(* PLC project Adressering.ecp, WAGO e!COCKPIT e!COCKPIT *)
(* stored: creationDateTime 2021-01-18T14:20:23.2110188, modificationDateTime 2021-01-18T11:51:27.6823754 *)

TYPE dtRomtype_11111111 : STRUCT
  RB601_V : BOOL;  (* Bevegelse *)
  RB601_HVAC : BOOL;  (* HVAC signal *)
  RT601_CT : REAL;  (* Rom temperatur *)
  RT601_SP_D : REAL;  (* Temperatur SP *)
  RT601_SP_S : REAL;  (* Temperatur SP standby *)
  RT601_SP_N : REAL;  (* Temperatur SP nattsenk *)
  RT601_SP_F : REAL;  (* Temperatur SP frostsikring *)
  RT601_CS : REAL;  (* Aktivt temperatur SP *)
  OPM : INT;  (* Rom modus *)
  OPM_CV : INT;  (* Rom modus verdi *)
  RY601_CV : REAL;  (* Co2 Nivaa *)
  RY601_SP : REAL;  (* Co2 SP *)
  RY601_MAN : BOOL;  (* Co2 Man mode *)
  RY601_OP : REAL;  (* Co2 paadrag *)
  LH601_OP : REAL;  (* Varmepaadrag *)
  LH601_MAN : BOOL;  (* Force LH *)
  LH601_CMD : BOOL;  (* LH601_CMD *)
  LC601_OP : REAL;  (* LC601_OP *)
  LC601_SP : REAL;  (* LC SP *)
  LC601_MAN : BOOL;  (* Force LC *)
  LC601_CMD : BOOL;  (* LC601_CMD *)
END_STRUCT;
END_TYPE

TYPE dtRomtype_22111111 : STRUCT
  RB601_V : BOOL;  (* Bevegelse *)
  RB602_V : BOOL;  (* Bevegelse *)
  RB601_HVAC : BOOL;  (* HVAC signal *)
  RB602_HVAC : BOOL;  (* HVAC signal *)
  RB600_HVAC : BOOL;  (* HVAC signal samlet *)
  RT601_CT : REAL;  (* Rom temperatur *)
  RT601_SP_D : REAL;  (* Temperatur SP *)
  RT601_SP_S : REAL;  (* Temperatur SP standby *)
  RT601_SP_N : REAL;  (* Temperatur SP nattsenk *)
  RT601_SP_F : REAL;  (* Temperatur SP frostsikring *)
  RT601_CS : REAL;  (* Aktivt temperatur SP *)
  OPM : INT;  (* Rom modus *)
  OPM_CV : INT;  (* Rom modus verdi *)
  RY601_CV : REAL;  (* Co2 Nivaa *)
  RY601_SP : REAL;  (* Co2 SP *)
  RY601_MAN : BOOL;  (* Co2 Man mode *)
  RY601_OP : REAL;  (* Co2 paadrag *)
  LH601_OP : REAL;  (* Varmepaadrag *)
  LH601_MAN : BOOL;  (* Force LH *)
  LH601_CMD : BOOL;  (* LH601_CMD *)
  LC601_OP : REAL;  (* LC601_OP *)
  LC601_SP : REAL;  (* LC SP *)
  LC601_MAN : BOOL;  (* Force LC *)
  LC601_CMD : BOOL;  (* LC601_CMD *)
END_STRUCT;
END_TYPE

TYPE dtRomtype_11211111 : STRUCT
  RB601_V : BOOL;  (* Bevegelse *)
  RB601_HVAC : BOOL;  (* HVAC signal *)
  RT601_CT : REAL;  (* Rom temperatur *)
  RT602_CT : REAL;  (* Rom temperatur *)
  RT600_CT : REAL;  (* Temperatur SP *)
  RT600_SP_D : REAL;  (* Temperatur SP *)
  RT600_SP_S : REAL;  (* Temperatur SP standby *)
  RT600_SP_N : REAL;  (* Temperatur SP nattsenk *)
  RT600_SP_F : REAL;  (* Temperatur SP frostsikring *)
  RT600_CS : REAL;  (* Aktivt temperatur SP *)
  OPM : INT;  (* Rom modus *)
  OPM_CV : INT;  (* Rom modus verdi *)
  RY601_CV : REAL;  (* Co2 Nivaa *)
  RY601_SP : REAL;  (* Co2 SP *)
  RY601_MAN : BOOL;  (* Co2 Man mode *)
  RY601_OP : REAL;  (* Co2 paadrag *)
  LH601_OP : REAL;  (* Varmepaadrag *)
  LH601_MAN : BOOL;  (* Force LH *)
  LH601_CMD : BOOL;  (* LH601_CMD *)
  LC601_OP : REAL;  (* LC601_OP *)
  LC601_SP : REAL;  (* LC SP *)
  LC601_MAN : BOOL;  (* Force LC *)
  LC601_CMD : BOOL;  (* LC601_CMD *)
END_STRUCT;
END_TYPE

TYPE dtRomtype_11121111 : STRUCT
  RB601_V : BOOL;  (* Bevegelse *)
  RB601_HVAC : BOOL;  (* HVAC signal *)
  RT601_CT : REAL;  (* Rom temperatur *)
  RT601_SP_D : REAL;  (* Temperatur SP *)
  RT601_SP_S : REAL;  (* Temperatur SP standby *)
  RT601_SP_N : REAL;  (* Temperatur SP nattsenk *)
  RT601_SP_F : REAL;  (* Temperatur SP frostsikring *)
  RT601_CS : REAL;  (* Aktivt temperatur SP *)
  OPM : INT;  (* Rom modus *)
  OPM_CV : INT;  (* Rom modus verdi *)
  RY601_CV : REAL;  (* Co2 Nivaa *)
  RY602_CV : REAL;  (* Co2 Nivaa *)
  RY600_CV : REAL;  (* Co2 gjennomsnitt *)
  RY600_SP : REAL;  (* Co2 SP *)
  RY600_MAN : BOOL;  (* Co2 Man mode *)
  RY600_OP : REAL;  (* Co2 paadrag *)
  LH601_OP : REAL;  (* Varmepaadrag *)
  LH601_MAN : BOOL;  (* Force LH *)
  LH601_CMD : BOOL;  (* LH601_CMD *)
  LC601_OP : REAL;  (* LC601_OP *)
  LC601_SP : REAL;  (* LC SP *)
  LC601_MAN : BOOL;  (* Force LC *)
  LC601_CMD : BOOL;  (* LC601_CMD *)
END_STRUCT;
END_TYPE

TYPE dtRomtype_11112111 : STRUCT
  RB601_V : BOOL;  (* Bevegelse *)
  RB601_HVAC : BOOL;  (* HVAC signal *)
  RT601_CT : REAL;  (* Rom temperatur *)
  RT601_SP_D : REAL;  (* Temperatur SP *)
  RT601_SP_S : REAL;  (* Temperatur SP standby *)
  RT601_SP_N : REAL;  (* Temperatur SP nattsenk *)
  RT601_SP_F : REAL;  (* Temperatur SP frostsikring *)
  RT601_CS : REAL;  (* Aktivt temperatur SP *)
  OPM : INT;  (* Rom modus *)
  OPM_CV : INT;  (* Rom modus verdi *)
  RY601_CV : REAL;  (* Co2 Nivaa *)
  RY601_SP : REAL;  (* Co2 SP *)
  RY601_MAN : BOOL;  (* Co2 Man mode *)
  RY601_OP : REAL;  (* Co2 paadrag *)
  LH601_OP : REAL;  (* Varmepaadrag *)
  LH602_OP : REAL;  (* Varmepaadrag *)
  LH601_MAN : BOOL;  (* Force LH *)
  LH601_CMD : BOOL;  (* LH601_CMD *)
  LC601_OP : REAL;  (* LC601_OP *)
  LC601_SP : REAL;  (* LC SP *)
  LC601_MAN : BOOL;  (* Force LC *)
  LC601_CMD : BOOL;  (* LC601_CMD *)
END_STRUCT;
END_TYPE

TYPE dtRomtype_11111211 : STRUCT
  RB601_V : BOOL;  (* Bevegelse *)
  RB601_HVAC : BOOL;  (* HVAC signal *)
  RT601_CT : REAL;  (* Rom temperatur *)
  RT601_SP_D : REAL;  (* Temperatur SP *)
  RT601_SP_S : REAL;  (* Temperatur SP standby *)
  RT601_SP_N : REAL;  (* Temperatur SP nattsenk *)
  RT601_SP_F : REAL;  (* Temperatur SP frostsikring *)
  RT601_CS : REAL;  (* Aktivt temperatur SP *)
  OPM : INT;  (* Rom modus *)
  OPM_CV : INT;  (* Rom modus verdi *)
  RY601_CV : REAL;  (* Co2 Nivaa *)
  RY601_SP : REAL;  (* Co2 SP *)
  RY601_MAN : BOOL;  (* Co2 Man mode *)
  RY601_OP : REAL;  (* Co2 paadrag *)
  LH601_OP : REAL;  (* Varmepaadrag *)
  LH601_MAN : BOOL;  (* Force LH *)
  LH601_CMD : BOOL;  (* LH601_CMD *)
  LH602_CMD : BOOL;  (* LH602_CMD *)
  LC601_OP : REAL;  (* LC601_OP *)
  LC601_SP : REAL;  (* LC SP *)
  LC601_MAN : BOOL;  (* Force LC *)
  LC601_CMD : BOOL;  (* LC601_CMD *)
END_STRUCT;
END_TYPE

TYPE dtRomtype_11111121 : STRUCT
  RB601_V : BOOL;  (* Bevegelse *)
  RB601_HVAC : BOOL;  (* HVAC signal *)
  RT601_CT : REAL;  (* Rom temperatur *)
  RT601_SP_D : REAL;  (* Temperatur SP *)
  RT601_SP_S : REAL;  (* Temperatur SP standby *)
  RT601_SP_N : REAL;  (* Temperatur SP nattsenk *)
  RT601_SP_F : REAL;  (* Temperatur SP frostsikring *)
  RT601_CS : REAL;  (* Aktivt temperatur SP *)
  OPM : INT;  (* Rom modus *)
  OPM_CV : INT;  (* Rom modus verdi *)
  RY601_CV : REAL;  (* Co2 Nivaa *)
  RY601_SP : REAL;  (* Co2 SP *)
  RY601_MAN : BOOL;  (* Co2 Man mode *)
  RY601_OP : REAL;  (* Co2 paadrag *)
  LH601_OP : REAL;  (* Varmepaadrag *)
  LH601_MAN : BOOL;  (* Force LH *)
  LH601_CMD : BOOL;  (* LH601_CMD *)
  LC601_OP : REAL;  (* LC601_OP *)
  LC602_OP : REAL;  (* LC602_OP *)
  LC601_SP : REAL;  (* LC SP *)
  LC601_MAN : BOOL;  (* Force LC *)
  LC601_CMD : BOOL;  (* LC601_CMD *)
END_STRUCT;
END_TYPE

TYPE dtRomtype_11111112 : STRUCT
  RB601_V : BOOL;  (* Bevegelse *)
  RB601_HVAC : BOOL;  (* HVAC signal *)
  RT601_CT : REAL;  (* Rom temperatur *)
  RT601_SP_D : REAL;  (* Temperatur SP *)
  RT601_SP_S : REAL;  (* Temperatur SP standby *)
  RT601_SP_N : REAL;  (* Temperatur SP nattsenk *)
  RT601_SP_F : REAL;  (* Temperatur SP frostsikring *)
  RT601_CS : REAL;  (* Aktivt temperatur SP *)
  OPM : INT;  (* Rom modus *)
  OPM_CV : INT;  (* Rom modus verdi *)
  RY601_CV : REAL;  (* Co2 Nivaa *)
  RY601_SP : REAL;  (* Co2 SP *)
  RY601_MAN : BOOL;  (* Co2 Man mode *)
  RY601_OP : REAL;  (* Co2 paadrag *)
  LH601_OP : REAL;  (* Varmepaadrag *)
  LH601_MAN : BOOL;  (* Force LH *)
  LH601_CMD : BOOL;  (* LH601_CMD *)
  LC601_OP : REAL;  (* LC601_OP *)
  LC601_SP : REAL;  (* LC SP *)
  LC601_MAN : BOOL;  (* Force LC *)
  LC601_CMD : BOOL;  (* LC601_CMD *)
  LC602_CMD : BOOL;  (* LC602_CMD *)
END_STRUCT;
END_TYPE

TYPE dtRomtype_11212111 : STRUCT
  RB601_V : BOOL;  (* Bevegelse *)
  RB601_HVAC : BOOL;  (* HVAC signal *)
  RT601_CT : REAL;  (* Rom temperatur *)
  RT602_CT : REAL;  (* Rom temperatur *)
  RT600_CT : REAL;  (* Temperatur SP *)
  RT600_SP_D : REAL;  (* Temperatur SP *)
  RT600_SP_S : REAL;  (* Temperatur SP standby *)
  RT600_SP_N : REAL;  (* Temperatur SP nattsenk *)
  RT600_SP_F : REAL;  (* Temperatur SP frostsikring *)
  RT600_CS : REAL;  (* Aktivt temperatur SP *)
  OPM : INT;  (* Rom modus *)
  OPM_CV : INT;  (* Rom modus verdi *)
  RY601_CV : REAL;  (* Co2 Nivaa *)
  RY601_SP : REAL;  (* Co2 SP *)
  RY601_MAN : BOOL;  (* Co2 Man mode *)
  RY601_OP : REAL;  (* Co2 paadrag *)
  LH601_OP : REAL;  (* Varmepaadrag *)
  LH602_OP : REAL;  (* Varmepaadrag *)
  LH601_MAN : BOOL;  (* Force LH *)
  LH601_CMD : BOOL;  (* LH601_CMD *)
  LC601_OP : REAL;  (* LC601_OP *)
  LC601_SP : REAL;  (* LC SP *)
  LC601_MAN : BOOL;  (* Force LC *)
  LC601_CMD : BOOL;  (* LC601_CMD *)
END_STRUCT;
END_TYPE

TYPE dtRomtype_11211211 : STRUCT
  RB601_V : BOOL;  (* Bevegelse *)
  RB601_HVAC : BOOL;  (* HVAC signal *)
  RT601_CT : REAL;  (* Rom temperatur *)
  RT602_CT : REAL;  (* Rom temperatur *)
  RT600_CT : REAL;  (* Temperatur SP *)
  RT600_SP_D : REAL;  (* Temperatur SP *)
  RT600_SP_S : REAL;  (* Temperatur SP standby *)
  RT600_SP_N : REAL;  (* Temperatur SP nattsenk *)
  RT600_SP_F : REAL;  (* Temperatur SP frostsikring *)
  RT600_CS : REAL;  (* Aktivt temperatur SP *)
  OPM : INT;  (* Rom modus *)
  OPM_CV : INT;  (* Rom modus verdi *)
  RY601_CV : REAL;  (* Co2 Nivaa *)
  RY601_SP : REAL;  (* Co2 SP *)
  RY601_MAN : BOOL;  (* Co2 Man mode *)
  RY601_OP : REAL;  (* Co2 paadrag *)
  LH601_OP : REAL;  (* Varmepaadrag *)
  LH601_MAN : BOOL;  (* Force LH *)
  LH601_CMD : BOOL;  (* LH601_CMD *)
  LH602_CMD : BOOL;  (* LH602_CMD *)
  LC601_OP : REAL;  (* LC601_OP *)
  LC601_SP : REAL;  (* LC SP *)
  LC601_MAN : BOOL;  (* Force LC *)
  LC601_CMD : BOOL;  (* LC601_CMD *)
END_STRUCT;
END_TYPE

TYPE dtRomtype_11211121 : STRUCT
  RB601_V : BOOL;  (* Bevegelse *)
  RB601_HVAC : BOOL;  (* HVAC signal *)
  RT601_CT : REAL;  (* Rom temperatur *)
  RT602_CT : REAL;  (* Rom temperatur *)
  RT600_CT : REAL;  (* Temperatur SP *)
  RT600_SP_D : REAL;  (* Temperatur SP *)
  RT600_SP_S : REAL;  (* Temperatur SP standby *)
  RT600_SP_N : REAL;  (* Temperatur SP nattsenk *)
  RT600_SP_F : REAL;  (* Temperatur SP frostsikring *)
  RT600_CS : REAL;  (* Aktivt temperatur SP *)
  OPM : INT;  (* Rom modus *)
  OPM_CV : INT;  (* Rom modus verdi *)
  RY601_CV : REAL;  (* Co2 Nivaa *)
  RY601_SP : REAL;  (* Co2 SP *)
  RY601_MAN : BOOL;  (* Co2 Man mode *)
  RY601_OP : REAL;  (* Co2 paadrag *)
  LH601_OP : REAL;  (* Varmepaadrag *)
  LH601_MAN : BOOL;  (* Force LH *)
  LH601_CMD : BOOL;  (* LH601_CMD *)
  LC601_OP : REAL;  (* LC601_OP *)
  LC602_OP : REAL;  (* LC602_OP *)
  LC601_SP : REAL;  (* LC SP *)
  LC601_MAN : BOOL;  (* Force LC *)
  LC601_CMD : BOOL;  (* LC601_CMD *)
END_STRUCT;
END_TYPE

TYPE dtRomtype_11211112 : STRUCT
  RB601_V : BOOL;  (* Bevegelse *)
  RB601_HVAC : BOOL;  (* HVAC signal *)
  RT601_CT : REAL;  (* Rom temperatur *)
  RT602_CT : REAL;  (* Rom temperatur *)
  RT600_CT : REAL;  (* Temperatur SP *)
  RT600_SP_D : REAL;  (* Temperatur SP *)
  RT600_SP_S : REAL;  (* Temperatur SP standby *)
  RT600_SP_N : REAL;  (* Temperatur SP nattsenk *)
  RT600_SP_F : REAL;  (* Temperatur SP frostsikring *)
  RT600_CS : REAL;  (* Aktivt temperatur SP *)
  OPM : INT;  (* Rom modus *)
  OPM_CV : INT;  (* Rom modus verdi *)
  RY601_CV : REAL;  (* Co2 Nivaa *)
  RY601_SP : REAL;  (* Co2 SP *)
  RY601_MAN : BOOL;  (* Co2 Man mode *)
  RY601_OP : REAL;  (* Co2 paadrag *)
  LH601_OP : REAL;  (* Varmepaadrag *)
  LH601_MAN : BOOL;  (* Force LH *)
  LH601_CMD : BOOL;  (* LH601_CMD *)
  LC601_OP : REAL;  (* LC601_OP *)
  LC601_SP : REAL;  (* LC SP *)
  LC601_MAN : BOOL;  (* Force LC *)
  LC601_CMD : BOOL;  (* LC601_CMD *)
  LC602_CMD : BOOL;  (* LC602_CMD *)
END_STRUCT;
END_TYPE

TYPE dtRomtype_11221111 : STRUCT
  RB601_V : BOOL;  (* Bevegelse *)
  RB601_HVAC : BOOL;  (* HVAC signal *)
  RT601_CT : REAL;  (* Rom temperatur *)
  RT602_CT : REAL;  (* Rom temperatur *)
  RT600_CT : REAL;  (* Temperatur SP *)
  RT600_SP_D : REAL;  (* Temperatur SP *)
  RT600_SP_S : REAL;  (* Temperatur SP standby *)
  RT600_SP_N : REAL;  (* Temperatur SP nattsenk *)
  RT600_SP_F : REAL;  (* Temperatur SP frostsikring *)
  RT600_CS : REAL;  (* Aktivt temperatur SP *)
  OPM : INT;  (* Rom modus *)
  OPM_CV : INT;  (* Rom modus verdi *)
  RY601_CV : REAL;  (* Co2 Nivaa *)
  RY602_CV : REAL;  (* Co2 Nivaa *)
  RY600_CV : REAL;  (* Co2 gjennomsnitt *)
  RY600_SP : REAL;  (* Co2 SP *)
  RY600_MAN : BOOL;  (* Co2 Man mode *)
  RY600_OP : REAL;  (* Co2 paadrag *)
  LH601_OP : REAL;  (* Varmepaadrag *)
  LH601_MAN : BOOL;  (* Force LH *)
  LH601_CMD : BOOL;  (* LH601_CMD *)
  LC601_OP : REAL;  (* LC601_OP *)
  LC601_SP : REAL;  (* LC SP *)
  LC601_MAN : BOOL;  (* Force LC *)
  LC601_CMD : BOOL;  (* LC601_CMD *)
END_STRUCT;
END_TYPE

TYPE dtRomtype_11222222 : STRUCT
  RB601_V : BOOL;  (* Bevegelse *)
  RB601_HVAC : BOOL;  (* HVAC signal *)
  RT601_CT : REAL;  (* Rom temperatur *)
  RT602_CT : REAL;  (* Rom temperatur *)
  RT600_CT : REAL;  (* Temperatur SP *)
  RT600_SP_D : REAL;  (* Temperatur SP *)
  RT600_SP_S : REAL;  (* Temperatur SP standby *)
  RT600_SP_N : REAL;  (* Temperatur SP nattsenk *)
  RT600_SP_F : REAL;  (* Temperatur SP frostsikring *)
  RT600_CS : REAL;  (* Aktivt temperatur SP *)
  OPM : INT;  (* Rom modus *)
  OPM_CV : INT;  (* Rom modus verdi *)
  RY601_CV : REAL;  (* Co2 Nivaa *)
  RY602_CV : REAL;  (* Co2 Nivaa *)
  RY600_CV : REAL;  (* Co2 gjennomsnitt *)
  RY600_SP : REAL;  (* Co2 SP *)
  RY600_MAN : BOOL;  (* Co2 Man mode *)
  RY600_OP : REAL;  (* Co2 paadrag *)
  LH601_OP : REAL;  (* Varmepaadrag *)
  LH602_OP : REAL;  (* Varmepaadrag *)
  LH601_MAN : BOOL;  (* Force LH *)
  LH601_CMD : BOOL;  (* LH601_CMD *)
  LH602_CMD : BOOL;  (* LH602_CMD *)
  LC601_OP : REAL;  (* LC601_OP *)
  LC602_OP : REAL;  (* LC602_OP *)
  LC601_SP : REAL;  (* LC SP *)
  LC601_MAN : BOOL;  (* Force LC *)
  LC601_CMD : BOOL;  (* LC601_CMD *)
  LC602_CMD : BOOL;  (* LC602_CMD *)
END_STRUCT;
END_TYPE

TYPE dtRomtype_22222222 : STRUCT
  RB601_V : BOOL;  (* Bevegelse *)
  RB602_V : BOOL;  (* Bevegelse *)
  RB601_HVAC : BOOL;  (* HVAC signal *)
  RB602_HVAC : BOOL;  (* HVAC signal *)
  RB600_HVAC : BOOL;  (* HVAC signal samlet *)
  RT601_CT : REAL;  (* Rom temperatur *)
  RT602_CT : REAL;  (* Rom temperatur *)
  RT600_CT : REAL;  (* Temperatur SP *)
  RT600_SP_D : REAL;  (* Temperatur SP *)
  RT600_SP_S : REAL;  (* Temperatur SP standby *)
  RT600_SP_N : REAL;  (* Temperatur SP nattsenk *)
  RT600_SP_F : REAL;  (* Temperatur SP frostsikring *)
  RT600_CS : REAL;  (* Aktivt temperatur SP *)
  OPM : INT;  (* Rom modus *)
  OPM_CV : INT;  (* Rom modus verdi *)
  RY601_CV : REAL;  (* Co2 Nivaa *)
  RY602_CV : REAL;  (* Co2 Nivaa *)
  RY600_CV : REAL;  (* Co2 gjennomsnitt *)
  RY600_SP : REAL;  (* Co2 SP *)
  RY600_MAN : BOOL;  (* Co2 Man mode *)
  RY600_OP : REAL;  (* Co2 paadrag *)
  LH601_OP : REAL;  (* Varmepaadrag *)
  LH602_OP : REAL;  (* Varmepaadrag *)
  LH601_MAN : BOOL;  (* Force LH *)
  LH601_CMD : BOOL;  (* LH601_CMD *)
  LH602_CMD : BOOL;  (* LH602_CMD *)
  LC601_OP : REAL;  (* LC601_OP *)
  LC602_OP : REAL;  (* LC602_OP *)
  LC601_SP : REAL;  (* LC SP *)
  LC601_MAN : BOOL;  (* Force LC *)
  LC601_CMD : BOOL;  (* LC601_CMD *)
  LC602_CMD : BOOL;  (* LC602_CMD *)
END_STRUCT;
END_TYPE

TYPE dtRomtype_22022222 : STRUCT
  RB601_V : BOOL;  (* Bevegelse *)
  RB602_V : BOOL;  (* Bevegelse *)
  RB601_HVAC : BOOL;  (* HVAC signal *)
  RB602_HVAC : BOOL;  (* HVAC signal *)
  RB600_HVAC : BOOL;  (* HVAC signal samlet *)
  RY601_CV : REAL;  (* Co2 Nivaa *)
  RY602_CV : REAL;  (* Co2 Nivaa *)
  RY600_CV : REAL;  (* Co2 gjennomsnitt *)
  RY600_SP : REAL;  (* Co2 SP *)
  RY600_MAN : BOOL;  (* Co2 Man mode *)
  RY600_OP : REAL;  (* Co2 paadrag *)
  LH601_OP : REAL;  (* Varmepaadrag *)
  LH602_OP : REAL;  (* Varmepaadrag *)
  LH601_MAN : BOOL;  (* Force LH *)
  LH601_CMD : BOOL;  (* LH601_CMD *)
  LH602_CMD : BOOL;  (* LH602_CMD *)
  LC601_OP : REAL;  (* LC601_OP *)
  LC602_OP : REAL;  (* LC602_OP *)
  LC601_SP : REAL;  (* LC SP *)
  LC601_MAN : BOOL;  (* Force LC *)
  LC601_CMD : BOOL;  (* LC601_CMD *)
  LC602_CMD : BOOL;  (* LC602_CMD *)
END_STRUCT;
END_TYPE

{attribute 'qualified_only'}
VAR_GLOBAL  (* STLV59_563 *)
  STLV59_A_563_RB001_HVAC : BOOL;  (* HVAC signal for PLS *)
  STLV59_A_563_KNX_Card_1_Status : BOOL;  (* KNX kort 1 status *)
  STLV59_A_563_001 : dtRomtype_11111111;  (* Test 1 *)
  STLV59_A_563_002 : dtRomtype_22111111;  (* Test 2 *)
  STLV59_A_563_003 : dtRomtype_11211111;  (* Test 3 *)
  STLV59_A_563_004 : dtRomtype_11121111;  (* Test 4 *)
  STLV59_A_563_005 : dtRomtype_11112111;  (* Test 5 *)
  STLV59_A_563_006 : dtRomtype_11111211;  (* Test 6 *)
  STLV59_A_563_007 : dtRomtype_11111121;  (* Test 7 *)
  STLV59_A_563_008 : dtRomtype_11111112;  (* Test 8 *)
  STLV59_A_563_009 : dtRomtype_11212111;  (* Test 9 *)
  STLV59_A_563_010 : dtRomtype_11211211;  (* Test 10 *)
  STLV59_A_563_011 : dtRomtype_11211121;  (* Test 11 *)
  STLV59_A_563_012 : dtRomtype_11211112;  (* Test 12 *)
  STLV59_A_563_013 : dtRomtype_11221111;  (* Test 13 *)
  STLV59_A_563_014 : dtRomtype_11222222;  (* Test 14 *)
  STLV59_A_563_015 : dtRomtype_22222222;  (* Test 15 *)
  STLV59_A_563_016 : dtRomtype_22022222;  (* Test 16 *)
END_VAR

FUNCTION_BLOCK fbRomtype_11111111
  VAR_INPUT
    RB601_HVAC : BOOL;
    RT601_CT : REAL;
    RT601_SP_D : REAL;
    RT601_SP_S : REAL;
    RT601_SP_N : REAL;
    RT601_SP_F : REAL;
    OPM : INT;
    RY601_CV : REAL;
    RY601_SP : REAL;
    RY601_MAN : BOOL;
    LH601_MAN : BOOL;
    LC601_SP : REAL;
    LC601_MAN : BOOL;
  END_VAR
  VAR
    RY601_PID_Man : BOOL;  (* Co2 regulering *)
    RY601_PID_ManVal : REAL;
    RY601_PID : fbSE_PID;
    RY601_PID_Kp : REAL := 1;  (* PID Luft rom. Forsterkning *)
    RY601_PID_Ti : REAL := 10;  (* PID luft rom. I-tid *)
    RY601_PID_Td : REAL;  (* PID luft rom. D-tid *)
    RY601_PID_Zero : REAL;  (* PID luft rom. 0-punkt *)
    RY601_PID_Max : REAL := 2000;  (* PID luft rom. Max verdi ppm *)
    RY601_PID_fMan : REAL := 100;  (* PID varme rom. Manuelt kjoeling *)
    LH601_PID : fbSE_PID;  (* PID varme rom *)
    LH601_PID_Kp : REAL := 1;  (* PID varme rom. Forsterkning *)
    LH601_PID_Ti : REAL := 10;  (* PID varme rom. I-tid *)
    LH601_PID_Td : REAL;  (* PID varme rom. D-tid *)
    LH601_PID_fMan : REAL := 100;  (* PID varme rom. Manuelt paadrag *)
    LH601_T : fbSE_Hyst;  (* Termostat varme rom *)
    LH601_T_On : REAL := 0.5;
    LH601_T_Off : REAL := 0.1;
    LC601_PID : fbSE_PID;  (* PID kjoeling rom *)
    LC601_PID_Kp : REAL := 1;  (* PID kjoeling rom. Forsterkning *)
    LC601_PID_Ti : REAL := 10;  (* PID kjoeling rom. I-tid *)
    LC601_PID_Td : REAL;  (* PID kjoeling rom. D-tid *)
    LC601_PID_fMan : REAL := 100;  (* PID varme rom. Manuelt kjoeling *)
    LC601_T : fbSE_Hyst;  (* Termostat kjoeling rom *)
    LC601_T_On : REAL := 0.5;
    LC601_T_Off : REAL := 0.1;
  END_VAR
  VAR_OUTPUT
    OPM_CV : INT;
    RT601_CS : REAL;
    RY601_OP : REAL;
    LH601_OP : REAL;
    LH601_CMD : BOOL;
    LC601_OP : REAL;
    LC601_CMD : BOOL;
  END_VAR

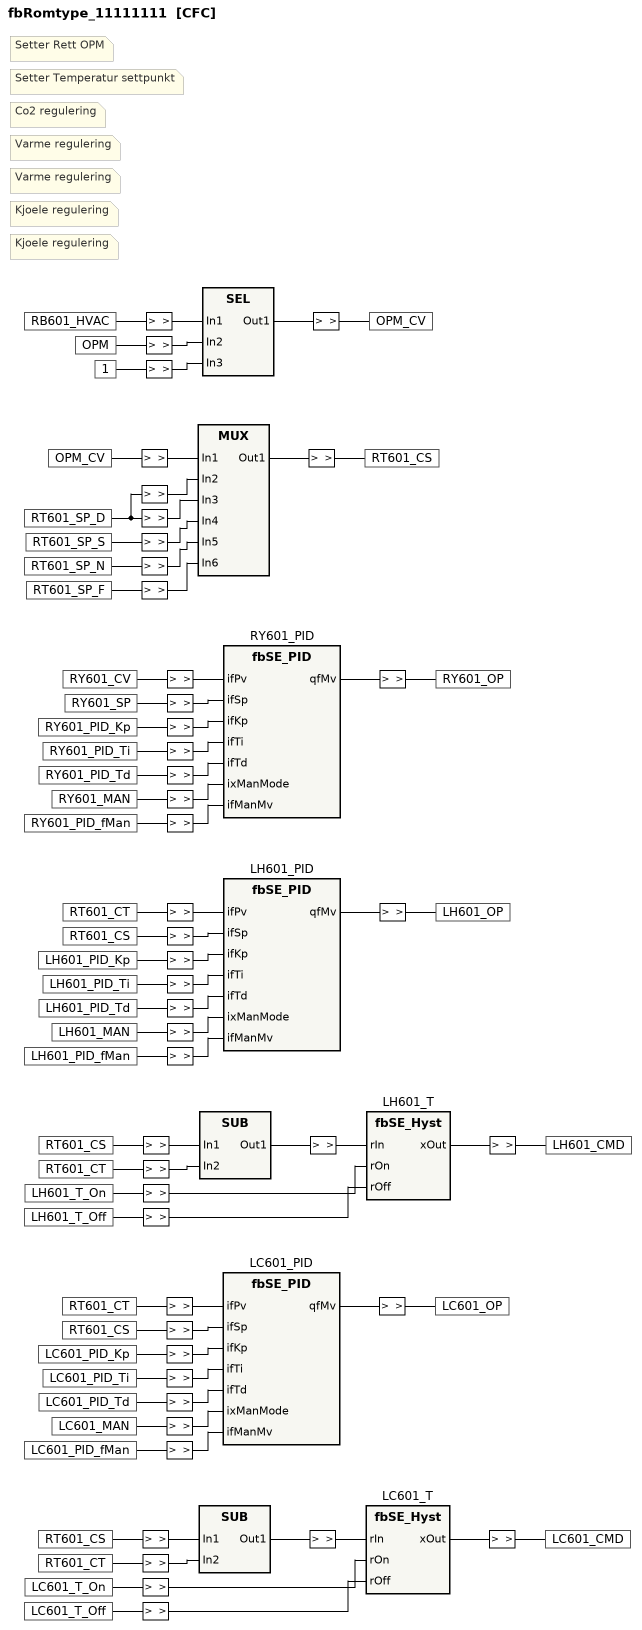
(* CFC diagram, written out as Structured Text *)
(* Setter Rett OPM *)
OPM_CV := SEL(RB601_HVAC, OPM, 1);
(* Setter Temperatur settpunkt *)
RT601_CS := MUX(OPM_CV, RT601_SP_D, RT601_SP_D, RT601_SP_S, RT601_SP_N, RT601_SP_F);
(* Co2 regulering *)
RY601_PID(ifPv := RY601_CV, ifSp := RY601_SP, ifKp := RY601_PID_Kp, ifTi := RY601_PID_Ti, ifTd := RY601_PID_Td, ixManMode := RY601_MAN, ifManMv := RY601_PID_fMan);
RY601_OP := RY601_PID.qfMv;
(* Varme regulering *)
LH601_PID(ifPv := RT601_CT, ifSp := RT601_CS, ifKp := LH601_PID_Kp, ifTi := LH601_PID_Ti, ifTd := LH601_PID_Td, ixManMode := LH601_MAN, ifManMv := LH601_PID_fMan);
LH601_OP := LH601_PID.qfMv;
(* Varme regulering *)
LH601_T(rIn := RT601_CS - RT601_CT, rOn := LH601_T_On, rOff := LH601_T_Off);
LH601_CMD := LH601_T.xOut;
(* Kjoele regulering *)
LC601_PID(ifPv := RT601_CT, ifSp := RT601_CS, ifKp := LC601_PID_Kp, ifTi := LC601_PID_Ti, ifTd := LC601_PID_Td, ixManMode := LC601_MAN, ifManMv := LC601_PID_fMan);
LC601_OP := LC601_PID.qfMv;
(* Kjoele regulering *)
LC601_T(rIn := RT601_CS - RT601_CT, rOn := LC601_T_On, rOff := LC601_T_Off);
LC601_CMD := LC601_T.xOut;
END_FUNCTION_BLOCK

FUNCTION_BLOCK fbRomtype_22111111
  VAR_INPUT
    RB601_HVAC : BOOL;
    RB602_HVAC : BOOL;
    RT601_CT : REAL;
    RT601_SP_D : REAL;
    RT601_SP_S : REAL;
    RT601_SP_N : REAL;
    RT601_SP_F : REAL;
    OPM : INT;
    RY601_CV : REAL;
    RY601_SP : REAL;
    RY601_MAN : BOOL;
    LH601_MAN : BOOL;
    LC601_SP : REAL;
    LC601_MAN : BOOL;
  END_VAR
  VAR
    RY601_PID_Man : BOOL;  (* Co2 regulering *)
    RY601_PID_ManVal : REAL;
    RY601_PID : fbSE_PID;
    RY601_PID_Kp : REAL := 1;  (* PID Luft rom. Forsterkning *)
    RY601_PID_Ti : REAL := 10;  (* PID luft rom. I-tid *)
    RY601_PID_Td : REAL;  (* PID luft rom. D-tid *)
    RY601_PID_Zero : REAL;  (* PID luft rom. 0-punkt *)
    RY601_PID_Max : REAL := 2000;  (* PID luft rom. Max verdi ppm *)
    RY601_PID_fMan : REAL := 100;  (* PID varme rom. Manuelt kjoeling *)
    LH601_PID : fbSE_PID;  (* PID varme rom *)
    LH601_PID_Kp : REAL := 1;  (* PID varme rom. Forsterkning *)
    LH601_PID_Ti : REAL := 10;  (* PID varme rom. I-tid *)
    LH601_PID_Td : REAL;  (* PID varme rom. D-tid *)
    LH601_PID_fMan : REAL := 100;  (* PID varme rom. Manuelt paadrag *)
    LH601_T : fbSE_Hyst;  (* Termostat varme rom *)
    LH601_T_On : REAL := 0.5;
    LH601_T_Off : REAL := 0.1;
    LC601_PID : fbSE_PID;  (* PID kjoeling rom *)
    LC601_PID_Kp : REAL := 1;  (* PID kjoeling rom. Forsterkning *)
    LC601_PID_Ti : REAL := 10;  (* PID kjoeling rom. I-tid *)
    LC601_PID_Td : REAL;  (* PID kjoeling rom. D-tid *)
    LC601_PID_fMan : REAL := 100;  (* PID varme rom. Manuelt kjoeling *)
    LC601_T : fbSE_Hyst;  (* Termostat kjoeling rom *)
    LC601_T_On : REAL := 0.5;
    LC601_T_Off : REAL := 0.1;
  END_VAR
  VAR_OUTPUT
    RB600_HVAC : BOOL;
    OPM_CV : INT;
    RT601_CS : REAL;
    RY601_OP : REAL;
    LH601_OP : REAL;
    LH601_CMD : BOOL;
    LC601_OP : REAL;
    LC601_CMD : BOOL;
  END_VAR
  VAR  (* added by the conversion: wires and edge detectors of the diagram *)
    _OR5_OUT : BOOL;
  END_VAR

(* CFC diagram, written out as Structured Text *)
(* Setter Rett OPM *)
_OR5_OUT := RB601_HVAC OR RB602_HVAC;
OPM_CV := SEL(_OR5_OUT, OPM, 1);
RB600_HVAC := _OR5_OUT;
(* Setter Temperatur settpunkt *)
RT601_CS := MUX(OPM_CV, RT601_SP_D, RT601_SP_D, RT601_SP_S, RT601_SP_N, RT601_SP_F);
(* Co2 regulering *)
RY601_PID(ifPv := RY601_CV, ifSp := RY601_SP, ifKp := RY601_PID_Kp, ifTi := RY601_PID_Ti, ifTd := RY601_PID_Td, ixManMode := RY601_MAN, ifManMv := RY601_PID_fMan);
RY601_OP := RY601_PID.qfMv;
(* Varme regulering *)
LH601_PID(ifPv := RT601_CT, ifSp := RT601_CS, ifKp := LH601_PID_Kp, ifTi := LH601_PID_Ti, ifTd := LH601_PID_Td, ixManMode := LH601_MAN, ifManMv := LH601_PID_fMan);
LH601_OP := LH601_PID.qfMv;
(* Varme regulering *)
LH601_T(rIn := RT601_CS - RT601_CT, rOn := LH601_T_On, rOff := LH601_T_Off);
LH601_CMD := LH601_T.xOut;
(* Kjoele regulering *)
LC601_PID(ifPv := RT601_CT, ifSp := RT601_CS, ifKp := LC601_PID_Kp, ifTi := LC601_PID_Ti, ifTd := LC601_PID_Td, ixManMode := LC601_MAN, ifManMv := LC601_PID_fMan);
LC601_OP := LC601_PID.qfMv;
(* Kjoele regulering *)
LC601_T(rIn := RT601_CS - RT601_CT, rOn := LC601_T_On, rOff := LC601_T_Off);
LC601_CMD := LC601_T.xOut;
END_FUNCTION_BLOCK

FUNCTION_BLOCK fbRomtype_11211111
  VAR_INPUT
    RB601_HVAC : BOOL;
    RT601_CT : REAL;
    RT602_CT : REAL;
    RT600_SP_D : REAL;
    RT600_SP_S : REAL;
    RT600_SP_N : REAL;
    RT600_SP_F : REAL;
    OPM : INT;
    RY601_CV : REAL;
    RY601_SP : REAL;
    RY601_MAN : BOOL;
    LH600_MAN : BOOL;
    LC600_SP : REAL;
    LC600_MAN : BOOL;
  END_VAR
  VAR
    RY601_PID_Man : BOOL;  (* Co2 regulering *)
    RY601_PID_ManVal : REAL;
    RY601_PID : fbSE_PID;
    RY601_PID_Kp : REAL := 1;  (* PID Luft rom. Forsterkning *)
    RY601_PID_Ti : REAL := 10;  (* PID luft rom. I-tid *)
    RY601_PID_Td : REAL;  (* PID luft rom. D-tid *)
    RY601_PID_Zero : REAL;  (* PID luft rom. 0-punkt *)
    RY601_PID_Max : REAL := 2000;  (* PID luft rom. Max verdi ppm *)
    RY601_PID_fMan : REAL := 100;  (* PID varme rom. Manuelt kjoeling *)
    LH600_PID : fbSE_PID;  (* PID varme rom *)
    LH600_PID_Kp : REAL := 1;  (* PID varme rom. Forsterkning *)
    LH600_PID_Ti : REAL := 10;  (* PID varme rom. I-tid *)
    LH600_PID_Td : REAL;  (* PID varme rom. D-tid *)
    LH600_PID_fMan : REAL := 100;  (* PID varme rom. Manuelt paadrag *)
    LH600_T : fbSE_Hyst;  (* Termostat varme rom *)
    LH600_T_On : REAL := 0.5;
    LH600_T_Off : REAL := 0.1;
    LC600_PID : fbSE_PID;  (* PID kjoeling rom *)
    LC600_PID_Kp : REAL := 1;  (* PID kjoeling rom. Forsterkning *)
    LC600_PID_Ti : REAL := 10;  (* PID kjoeling rom. I-tid *)
    LC600_PID_Td : REAL;  (* PID kjoeling rom. D-tid *)
    LC600_PID_fMan : REAL := 100;  (* PID varme rom. Manuelt kjoeling *)
    LC600_T : fbSE_Hyst;  (* Termostat kjoeling rom *)
    LC600_T_On : REAL := 0.5;
    LC600_T_Off : REAL := 0.1;
  END_VAR
  VAR_OUTPUT
    OPM_CV : INT;
    RT600_CT : REAL;
    RT600_CS : REAL;
    RY601_OP : REAL;
    LH601_OP : REAL;
    LH601_CMD : BOOL;
    LC601_OP : REAL;
    LC601_CMD : BOOL;
  END_VAR
  VAR  (* added by the conversion: wires and edge detectors of the diagram *)
    _ADD30_OUT : REAL;
    _DIV39_ENO : BOOL;
    _DIV39_OUT : REAL;
  END_VAR

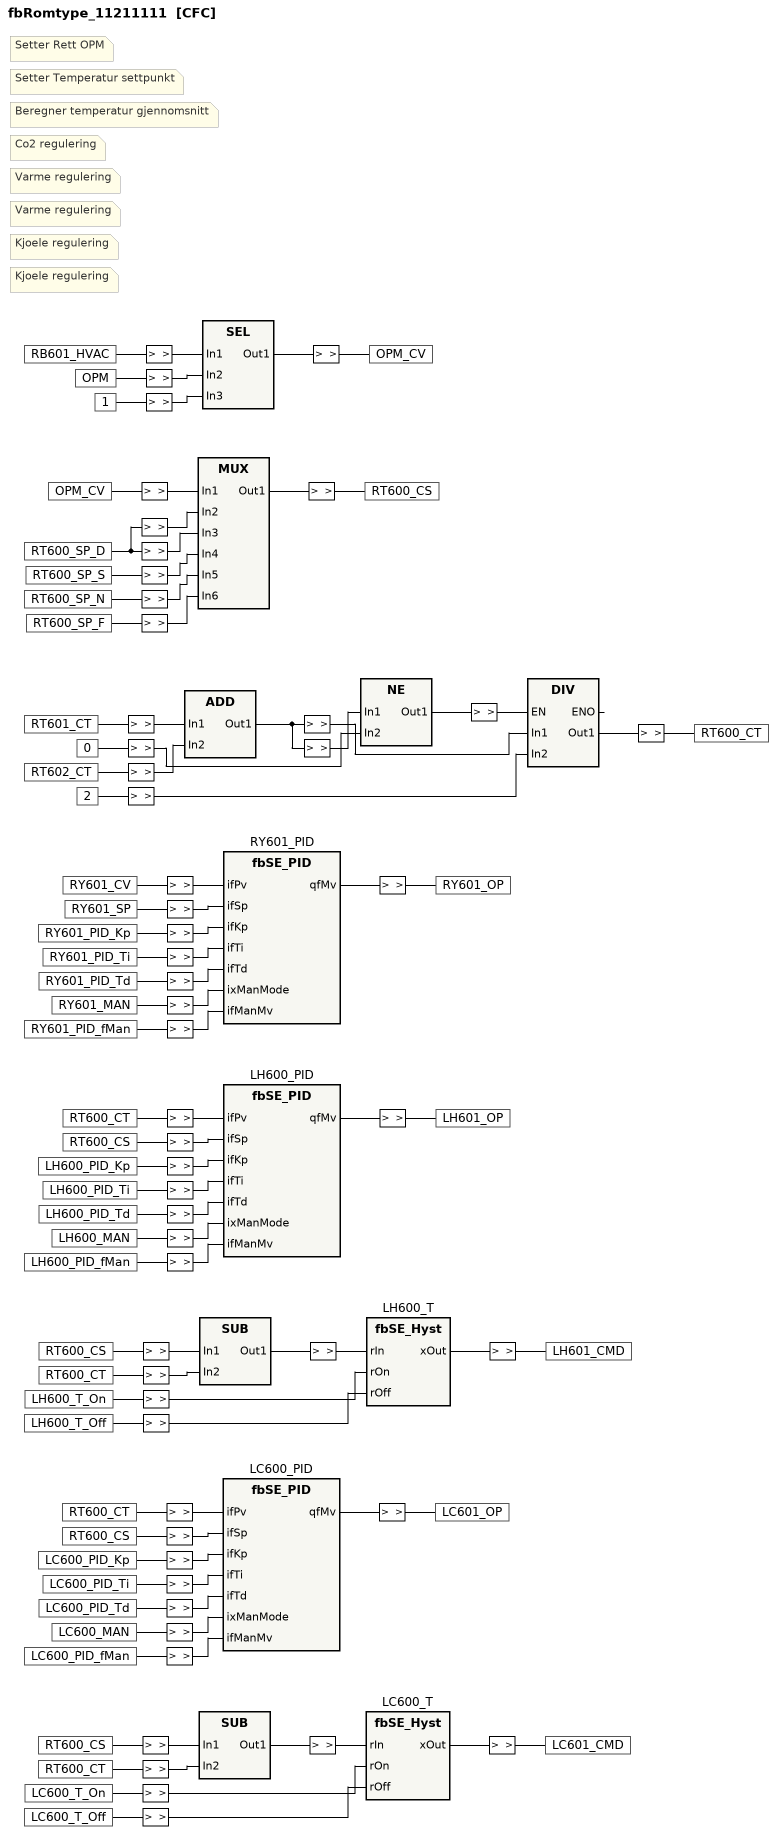
(* CFC diagram, written out as Structured Text *)
(* Setter Rett OPM *)
OPM_CV := SEL(RB601_HVAC, OPM, 1);
(* Setter Temperatur settpunkt *)
RT600_CS := MUX(OPM_CV, RT600_SP_D, RT600_SP_D, RT600_SP_S, RT600_SP_N, RT600_SP_F);
(* Beregner temperatur gjennomsnitt *)
_ADD30_OUT := RT601_CT + RT602_CT;
_DIV39_OUT := DIV(EN := _ADD30_OUT <> 0, IN1 := _ADD30_OUT, IN2 := 2, ENO => _DIV39_ENO);
IF _DIV39_ENO THEN RT600_CT := _DIV39_OUT; END_IF;
(* Co2 regulering *)
RY601_PID(ifPv := RY601_CV, ifSp := RY601_SP, ifKp := RY601_PID_Kp, ifTi := RY601_PID_Ti, ifTd := RY601_PID_Td, ixManMode := RY601_MAN, ifManMv := RY601_PID_fMan);
RY601_OP := RY601_PID.qfMv;
(* Varme regulering *)
LH600_PID(ifPv := RT600_CT, ifSp := RT600_CS, ifKp := LH600_PID_Kp, ifTi := LH600_PID_Ti, ifTd := LH600_PID_Td, ixManMode := LH600_MAN, ifManMv := LH600_PID_fMan);
LH601_OP := LH600_PID.qfMv;
(* Varme regulering *)
LH600_T(rIn := RT600_CS - RT600_CT, rOn := LH600_T_On, rOff := LH600_T_Off);
LH601_CMD := LH600_T.xOut;
(* Kjoele regulering *)
LC600_PID(ifPv := RT600_CT, ifSp := RT600_CS, ifKp := LC600_PID_Kp, ifTi := LC600_PID_Ti, ifTd := LC600_PID_Td, ixManMode := LC600_MAN, ifManMv := LC600_PID_fMan);
LC601_OP := LC600_PID.qfMv;
(* Kjoele regulering *)
LC600_T(rIn := RT600_CS - RT600_CT, rOn := LC600_T_On, rOff := LC600_T_Off);
LC601_CMD := LC600_T.xOut;
END_FUNCTION_BLOCK

FUNCTION_BLOCK fbRomtype_11121111
  VAR_INPUT
    RB601_HVAC : BOOL;
    RT601_CT : REAL;
    RT601_SP_D : REAL;
    RT601_SP_S : REAL;
    RT601_SP_N : REAL;
    RT601_SP_F : REAL;
    OPM : INT;
    RY601_CV : REAL;
    RY602_CV : REAL;
    RY600_SP : REAL;
    RY600_MAN : BOOL;
    LH601_MAN : BOOL;
    LC601_SP : REAL;
    LC601_MAN : BOOL;
  END_VAR
  VAR
    RY600_PID_Man : BOOL;  (* Co2 regulering *)
    RY600_PID_ManVal : REAL;
    RY600_PID : fbSE_PID;
    RY600_PID_Kp : REAL := 1;  (* PID Luft rom. Forsterkning *)
    RY600_PID_Ti : REAL := 10;  (* PID luft rom. I-tid *)
    RY600_PID_Td : REAL;  (* PID luft rom. D-tid *)
    RY600_PID_Zero : REAL;  (* PID luft rom. 0-punkt *)
    RY600_PID_Max : REAL := 2000;  (* PID luft rom. Max verdi ppm *)
    RY600_PID_fMan : REAL := 100;  (* PID varme rom. Manuelt kjoeling *)
    LH601_PID : fbSE_PID;  (* PID varme rom *)
    LH601_PID_Kp : REAL := 1;  (* PID varme rom. Forsterkning *)
    LH601_PID_Ti : REAL := 10;  (* PID varme rom. I-tid *)
    LH601_PID_Td : REAL;  (* PID varme rom. D-tid *)
    LH601_PID_fMan : REAL := 100;  (* PID varme rom. Manuelt paadrag *)
    LH601_T : fbSE_Hyst;  (* Termostat varme rom *)
    LH601_T_On : REAL := 0.5;
    LH601_T_Off : REAL := 0.1;
    LC601_PID : fbSE_PID;  (* PID kjoeling rom *)
    LC601_PID_Kp : REAL := 1;  (* PID kjoeling rom. Forsterkning *)
    LC601_PID_Ti : REAL := 10;  (* PID kjoeling rom. I-tid *)
    LC601_PID_Td : REAL;  (* PID kjoeling rom. D-tid *)
    LC601_PID_fMan : REAL := 100;  (* PID varme rom. Manuelt kjoeling *)
    LC601_T : fbSE_Hyst;  (* Termostat kjoeling rom *)
    LC601_T_On : REAL := 0.5;
    LC601_T_Off : REAL := 0.1;
  END_VAR
  VAR_OUTPUT
    OPM_CV : INT;
    RT601_CS : REAL;
    RY600_CV : REAL;
    RY600_OP : REAL;
    LH601_OP : REAL;
    LH601_CMD : BOOL;
    LC601_OP : REAL;
    LC601_CMD : BOOL;
  END_VAR
  VAR  (* added by the conversion: wires and edge detectors of the diagram *)
    _ADD30_OUT : REAL;
    _DIV39_ENO : BOOL;
    _DIV39_OUT : REAL;
  END_VAR

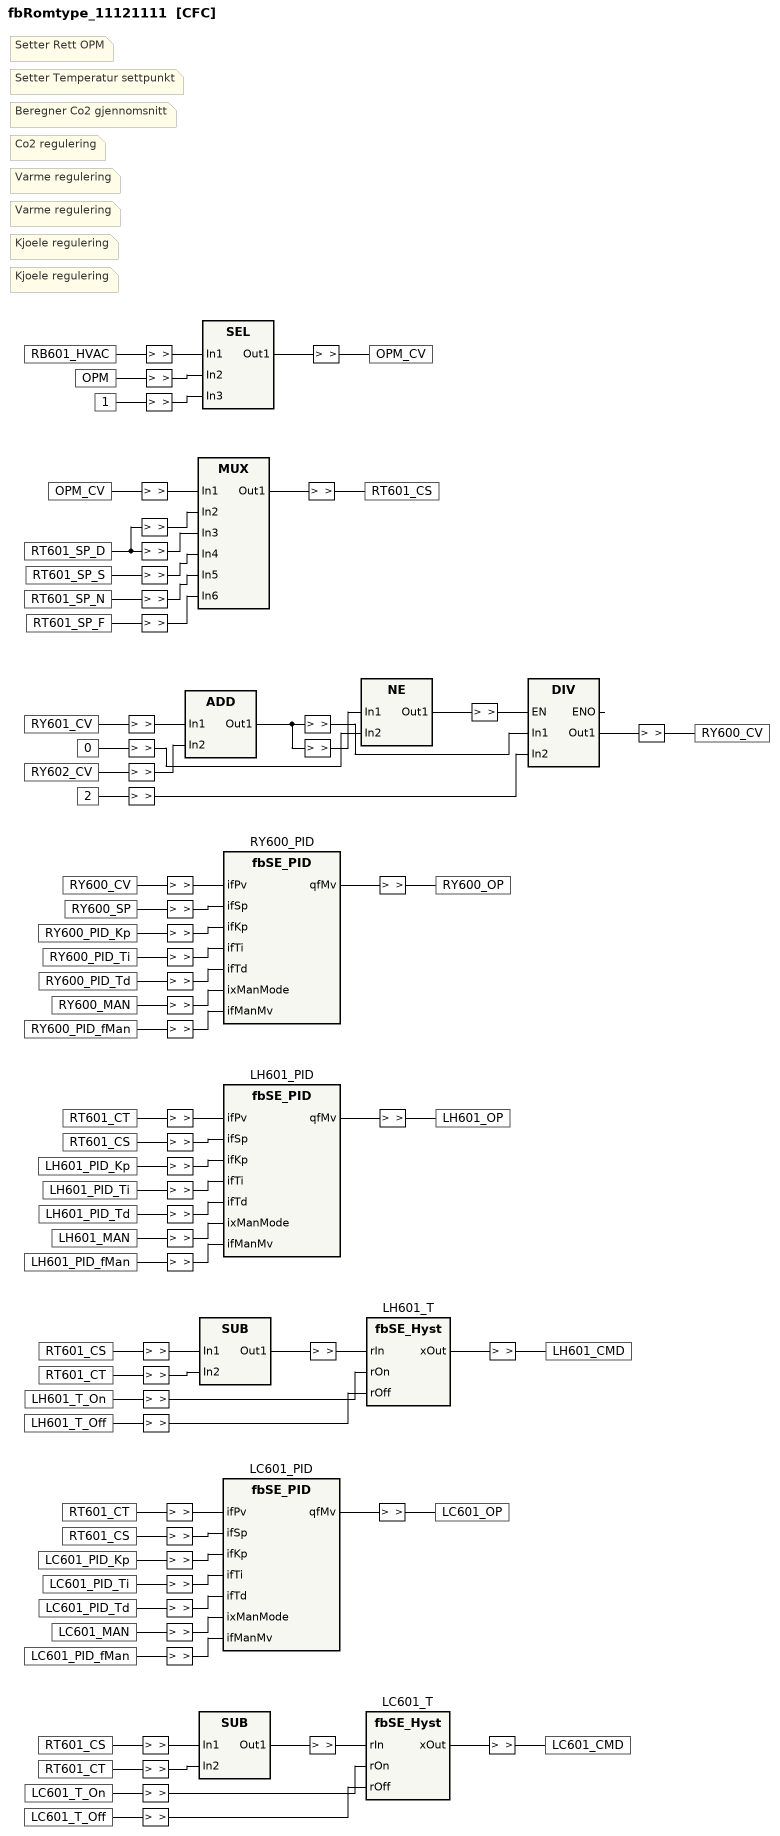
(* CFC diagram, written out as Structured Text *)
(* Setter Rett OPM *)
OPM_CV := SEL(RB601_HVAC, OPM, 1);
(* Setter Temperatur settpunkt *)
RT601_CS := MUX(OPM_CV, RT601_SP_D, RT601_SP_D, RT601_SP_S, RT601_SP_N, RT601_SP_F);
(* Beregner Co2 gjennomsnitt *)
_ADD30_OUT := RY601_CV + RY602_CV;
_DIV39_OUT := DIV(EN := _ADD30_OUT <> 0, IN1 := _ADD30_OUT, IN2 := 2, ENO => _DIV39_ENO);
IF _DIV39_ENO THEN RY600_CV := _DIV39_OUT; END_IF;
(* Co2 regulering *)
RY600_PID(ifPv := RY600_CV, ifSp := RY600_SP, ifKp := RY600_PID_Kp, ifTi := RY600_PID_Ti, ifTd := RY600_PID_Td, ixManMode := RY600_MAN, ifManMv := RY600_PID_fMan);
RY600_OP := RY600_PID.qfMv;
(* Varme regulering *)
LH601_PID(ifPv := RT601_CT, ifSp := RT601_CS, ifKp := LH601_PID_Kp, ifTi := LH601_PID_Ti, ifTd := LH601_PID_Td, ixManMode := LH601_MAN, ifManMv := LH601_PID_fMan);
LH601_OP := LH601_PID.qfMv;
(* Varme regulering *)
LH601_T(rIn := RT601_CS - RT601_CT, rOn := LH601_T_On, rOff := LH601_T_Off);
LH601_CMD := LH601_T.xOut;
(* Kjoele regulering *)
LC601_PID(ifPv := RT601_CT, ifSp := RT601_CS, ifKp := LC601_PID_Kp, ifTi := LC601_PID_Ti, ifTd := LC601_PID_Td, ixManMode := LC601_MAN, ifManMv := LC601_PID_fMan);
LC601_OP := LC601_PID.qfMv;
(* Kjoele regulering *)
LC601_T(rIn := RT601_CS - RT601_CT, rOn := LC601_T_On, rOff := LC601_T_Off);
LC601_CMD := LC601_T.xOut;
END_FUNCTION_BLOCK

FUNCTION_BLOCK fbRomtype_11112111
  VAR_INPUT
    RB601_HVAC : BOOL;
    RT601_CT : REAL;
    RT601_SP_D : REAL;
    RT601_SP_S : REAL;
    RT601_SP_N : REAL;
    RT601_SP_F : REAL;
    OPM : INT;
    RY601_CV : REAL;
    RY601_SP : REAL;
    RY601_MAN : BOOL;
    LH601_MAN : BOOL;
    LC601_SP : REAL;
    LC601_MAN : BOOL;
  END_VAR
  VAR
    RY601_PID_Man : BOOL;  (* Co2 regulering *)
    RY601_PID_ManVal : REAL;
    RY601_PID : fbSE_PID;
    RY601_PID_Kp : REAL := 1;  (* PID Luft rom. Forsterkning *)
    RY601_PID_Ti : REAL := 10;  (* PID luft rom. I-tid *)
    RY601_PID_Td : REAL;  (* PID luft rom. D-tid *)
    RY601_PID_Zero : REAL;  (* PID luft rom. 0-punkt *)
    RY601_PID_Max : REAL := 2000;  (* PID luft rom. Max verdi ppm *)
    RY601_PID_fMan : REAL := 100;  (* PID varme rom. Manuelt kjoeling *)
    LH601_PID : fbSE_PID;  (* PID varme rom *)
    LH601_PID_Kp : REAL := 1;  (* PID varme rom. Forsterkning *)
    LH601_PID_Ti : REAL := 10;  (* PID varme rom. I-tid *)
    LH601_PID_Td : REAL;  (* PID varme rom. D-tid *)
    LH601_PID_fMan : REAL := 100;  (* PID varme rom. Manuelt paadrag *)
    LH601_T : fbSE_Hyst;  (* Termostat varme rom *)
    LH601_T_On : REAL := 0.5;
    LH601_T_Off : REAL := 0.1;
    LC601_PID : fbSE_PID;  (* PID kjoeling rom *)
    LC601_PID_Kp : REAL := 1;  (* PID kjoeling rom. Forsterkning *)
    LC601_PID_Ti : REAL := 10;  (* PID kjoeling rom. I-tid *)
    LC601_PID_Td : REAL;  (* PID kjoeling rom. D-tid *)
    LC601_PID_fMan : REAL := 100;  (* PID varme rom. Manuelt kjoeling *)
    LC601_T : fbSE_Hyst;  (* Termostat kjoeling rom *)
    LC601_T_On : REAL := 0.5;
    LC601_T_Off : REAL := 0.1;
  END_VAR
  VAR_OUTPUT
    OPM_CV : INT;
    RT601_CS : REAL;
    RY601_OP : REAL;
    LH601_OP : REAL;
    LH602_OP : REAL;
    LH601_CMD : BOOL;
    LC601_OP : REAL;
    LC601_CMD : BOOL;
  END_VAR

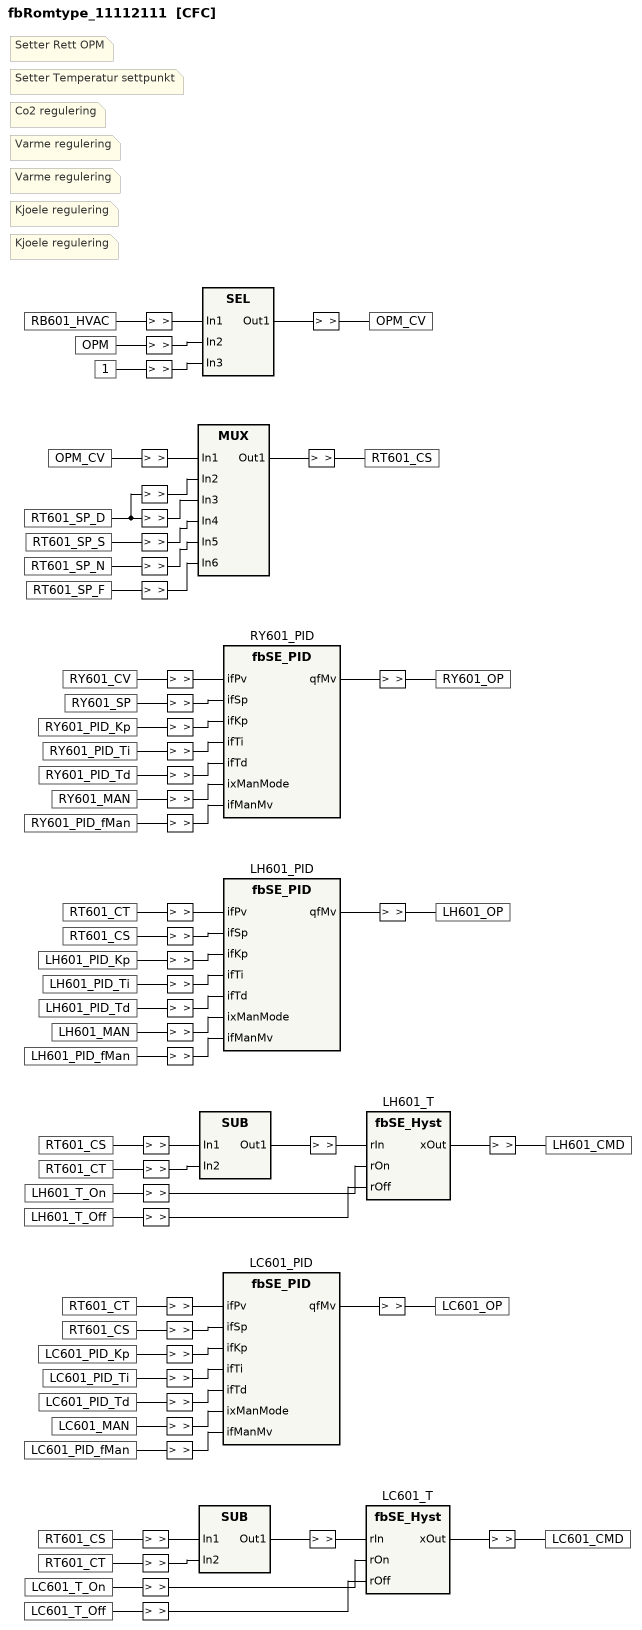
(* CFC diagram, written out as Structured Text *)
(* Setter Rett OPM *)
OPM_CV := SEL(RB601_HVAC, OPM, 1);
(* Setter Temperatur settpunkt *)
RT601_CS := MUX(OPM_CV, RT601_SP_D, RT601_SP_D, RT601_SP_S, RT601_SP_N, RT601_SP_F);
(* Co2 regulering *)
RY601_PID(ifPv := RY601_CV, ifSp := RY601_SP, ifKp := RY601_PID_Kp, ifTi := RY601_PID_Ti, ifTd := RY601_PID_Td, ixManMode := RY601_MAN, ifManMv := RY601_PID_fMan);
RY601_OP := RY601_PID.qfMv;
(* Varme regulering *)
LH601_PID(ifPv := RT601_CT, ifSp := RT601_CS, ifKp := LH601_PID_Kp, ifTi := LH601_PID_Ti, ifTd := LH601_PID_Td, ixManMode := LH601_MAN, ifManMv := LH601_PID_fMan);
LH601_OP := LH601_PID.qfMv;
(* Varme regulering *)
LH601_T(rIn := RT601_CS - RT601_CT, rOn := LH601_T_On, rOff := LH601_T_Off);
LH601_CMD := LH601_T.xOut;
(* Kjoele regulering *)
LC601_PID(ifPv := RT601_CT, ifSp := RT601_CS, ifKp := LC601_PID_Kp, ifTi := LC601_PID_Ti, ifTd := LC601_PID_Td, ixManMode := LC601_MAN, ifManMv := LC601_PID_fMan);
LC601_OP := LC601_PID.qfMv;
(* Kjoele regulering *)
LC601_T(rIn := RT601_CS - RT601_CT, rOn := LC601_T_On, rOff := LC601_T_Off);
LC601_CMD := LC601_T.xOut;
END_FUNCTION_BLOCK

FUNCTION_BLOCK fbRomtype_11111211
  VAR_INPUT
    RB601_HVAC : BOOL;
    RT601_CT : REAL;
    RT601_SP_D : REAL;
    RT601_SP_S : REAL;
    RT601_SP_N : REAL;
    RT601_SP_F : REAL;
    OPM : INT;
    RY601_CV : REAL;
    RY601_SP : REAL;
    RY601_MAN : BOOL;
    LH601_MAN : BOOL;
    LC601_SP : REAL;
    LC601_MAN : BOOL;
  END_VAR
  VAR
    RY601_PID_Man : BOOL;  (* Co2 regulering *)
    RY601_PID_ManVal : REAL;
    RY601_PID : fbSE_PID;
    RY601_PID_Kp : REAL := 1;  (* PID Luft rom. Forsterkning *)
    RY601_PID_Ti : REAL := 10;  (* PID luft rom. I-tid *)
    RY601_PID_Td : REAL;  (* PID luft rom. D-tid *)
    RY601_PID_Zero : REAL;  (* PID luft rom. 0-punkt *)
    RY601_PID_Max : REAL := 2000;  (* PID luft rom. Max verdi ppm *)
    RY601_PID_fMan : REAL := 100;  (* PID varme rom. Manuelt kjoeling *)
    LH601_PID : fbSE_PID;  (* PID varme rom *)
    LH601_PID_Kp : REAL := 1;  (* PID varme rom. Forsterkning *)
    LH601_PID_Ti : REAL := 10;  (* PID varme rom. I-tid *)
    LH601_PID_Td : REAL;  (* PID varme rom. D-tid *)
    LH601_PID_fMan : REAL := 100;  (* PID varme rom. Manuelt paadrag *)
    LH601_T : fbSE_Hyst;  (* Termostat varme rom *)
    LH601_T_On : REAL := 0.5;
    LH601_T_Off : REAL := 0.1;
    LC601_PID : fbSE_PID;  (* PID kjoeling rom *)
    LC601_PID_Kp : REAL := 1;  (* PID kjoeling rom. Forsterkning *)
    LC601_PID_Ti : REAL := 10;  (* PID kjoeling rom. I-tid *)
    LC601_PID_Td : REAL;  (* PID kjoeling rom. D-tid *)
    LC601_PID_fMan : REAL := 100;  (* PID varme rom. Manuelt kjoeling *)
    LC601_T : fbSE_Hyst;  (* Termostat kjoeling rom *)
    LC601_T_On : REAL := 0.5;
    LC601_T_Off : REAL := 0.1;
  END_VAR
  VAR_OUTPUT
    OPM_CV : INT;
    RT601_CS : REAL;
    RY601_OP : REAL;
    LH601_OP : REAL;
    LH601_CMD : BOOL;
    LH602_CMD : BOOL;
    LC601_OP : REAL;
    LC601_CMD : BOOL;
  END_VAR

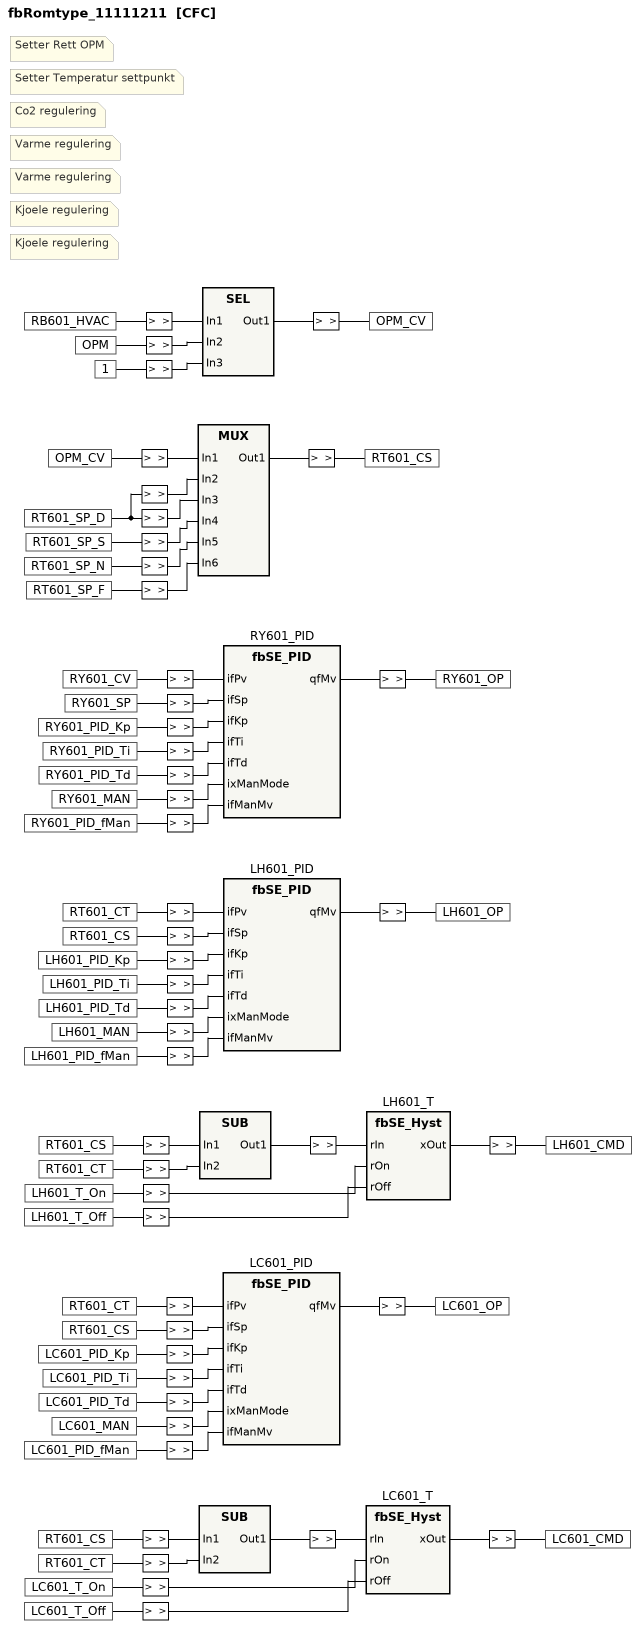
(* CFC diagram, written out as Structured Text *)
(* Setter Rett OPM *)
OPM_CV := SEL(RB601_HVAC, OPM, 1);
(* Setter Temperatur settpunkt *)
RT601_CS := MUX(OPM_CV, RT601_SP_D, RT601_SP_D, RT601_SP_S, RT601_SP_N, RT601_SP_F);
(* Co2 regulering *)
RY601_PID(ifPv := RY601_CV, ifSp := RY601_SP, ifKp := RY601_PID_Kp, ifTi := RY601_PID_Ti, ifTd := RY601_PID_Td, ixManMode := RY601_MAN, ifManMv := RY601_PID_fMan);
RY601_OP := RY601_PID.qfMv;
(* Varme regulering *)
LH601_PID(ifPv := RT601_CT, ifSp := RT601_CS, ifKp := LH601_PID_Kp, ifTi := LH601_PID_Ti, ifTd := LH601_PID_Td, ixManMode := LH601_MAN, ifManMv := LH601_PID_fMan);
LH601_OP := LH601_PID.qfMv;
(* Varme regulering *)
LH601_T(rIn := RT601_CS - RT601_CT, rOn := LH601_T_On, rOff := LH601_T_Off);
LH601_CMD := LH601_T.xOut;
(* Kjoele regulering *)
LC601_PID(ifPv := RT601_CT, ifSp := RT601_CS, ifKp := LC601_PID_Kp, ifTi := LC601_PID_Ti, ifTd := LC601_PID_Td, ixManMode := LC601_MAN, ifManMv := LC601_PID_fMan);
LC601_OP := LC601_PID.qfMv;
(* Kjoele regulering *)
LC601_T(rIn := RT601_CS - RT601_CT, rOn := LC601_T_On, rOff := LC601_T_Off);
LC601_CMD := LC601_T.xOut;
END_FUNCTION_BLOCK

FUNCTION_BLOCK fbRomtype_11111121
  VAR_INPUT
    RB601_HVAC : BOOL;
    RT601_CT : REAL;
    RT601_SP_D : REAL;
    RT601_SP_S : REAL;
    RT601_SP_N : REAL;
    RT601_SP_F : REAL;
    OPM : INT;
    RY601_CV : REAL;
    RY601_SP : REAL;
    RY601_MAN : BOOL;
    LH601_MAN : BOOL;
    LC601_SP : REAL;
    LC601_MAN : BOOL;
  END_VAR
  VAR
    RY601_PID_Man : BOOL;  (* Co2 regulering *)
    RY601_PID_ManVal : REAL;
    RY601_PID : fbSE_PID;
    RY601_PID_Kp : REAL := 1;  (* PID Luft rom. Forsterkning *)
    RY601_PID_Ti : REAL := 10;  (* PID luft rom. I-tid *)
    RY601_PID_Td : REAL;  (* PID luft rom. D-tid *)
    RY601_PID_Zero : REAL;  (* PID luft rom. 0-punkt *)
    RY601_PID_Max : REAL := 2000;  (* PID luft rom. Max verdi ppm *)
    RY601_PID_fMan : REAL := 100;  (* PID varme rom. Manuelt kjoeling *)
    LH601_PID : fbSE_PID;  (* PID varme rom *)
    LH601_PID_Kp : REAL := 1;  (* PID varme rom. Forsterkning *)
    LH601_PID_Ti : REAL := 10;  (* PID varme rom. I-tid *)
    LH601_PID_Td : REAL;  (* PID varme rom. D-tid *)
    LH601_PID_fMan : REAL := 100;  (* PID varme rom. Manuelt paadrag *)
    LH601_T : fbSE_Hyst;  (* Termostat varme rom *)
    LH601_T_On : REAL := 0.5;
    LH601_T_Off : REAL := 0.1;
    LC601_PID : fbSE_PID;  (* PID kjoeling rom *)
    LC601_PID_Kp : REAL := 1;  (* PID kjoeling rom. Forsterkning *)
    LC601_PID_Ti : REAL := 10;  (* PID kjoeling rom. I-tid *)
    LC601_PID_Td : REAL;  (* PID kjoeling rom. D-tid *)
    LC601_PID_fMan : REAL := 100;  (* PID varme rom. Manuelt kjoeling *)
    LC601_T : fbSE_Hyst;  (* Termostat kjoeling rom *)
    LC601_T_On : REAL := 0.5;
    LC601_T_Off : REAL := 0.1;
  END_VAR
  VAR_OUTPUT
    OPM_CV : INT;
    RT601_CS : REAL;
    RY601_OP : REAL;
    LH601_OP : REAL;
    LH601_CMD : BOOL;
    LC601_OP : REAL;
    LC602_OP : REAL;
    LC601_CMD : BOOL;
  END_VAR

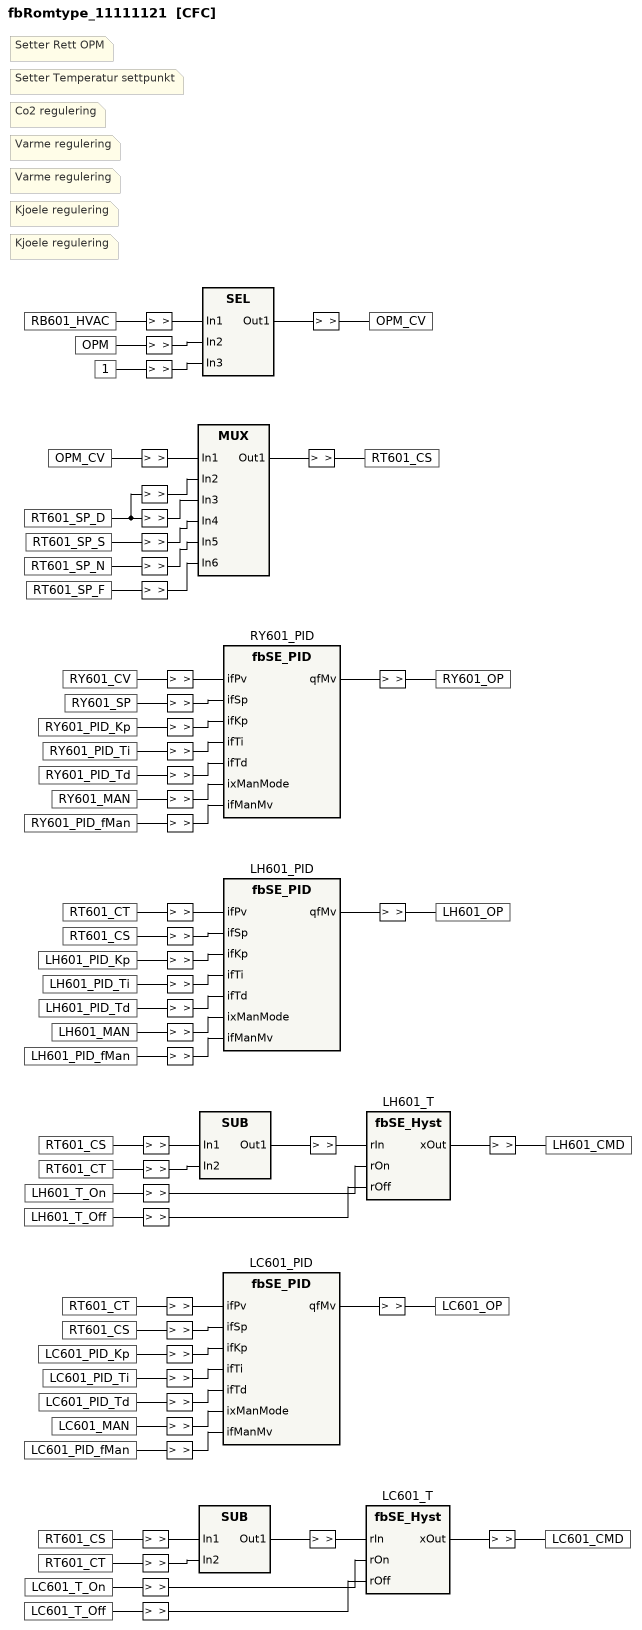
(* CFC diagram, written out as Structured Text *)
(* Setter Rett OPM *)
OPM_CV := SEL(RB601_HVAC, OPM, 1);
(* Setter Temperatur settpunkt *)
RT601_CS := MUX(OPM_CV, RT601_SP_D, RT601_SP_D, RT601_SP_S, RT601_SP_N, RT601_SP_F);
(* Co2 regulering *)
RY601_PID(ifPv := RY601_CV, ifSp := RY601_SP, ifKp := RY601_PID_Kp, ifTi := RY601_PID_Ti, ifTd := RY601_PID_Td, ixManMode := RY601_MAN, ifManMv := RY601_PID_fMan);
RY601_OP := RY601_PID.qfMv;
(* Varme regulering *)
LH601_PID(ifPv := RT601_CT, ifSp := RT601_CS, ifKp := LH601_PID_Kp, ifTi := LH601_PID_Ti, ifTd := LH601_PID_Td, ixManMode := LH601_MAN, ifManMv := LH601_PID_fMan);
LH601_OP := LH601_PID.qfMv;
(* Varme regulering *)
LH601_T(rIn := RT601_CS - RT601_CT, rOn := LH601_T_On, rOff := LH601_T_Off);
LH601_CMD := LH601_T.xOut;
(* Kjoele regulering *)
LC601_PID(ifPv := RT601_CT, ifSp := RT601_CS, ifKp := LC601_PID_Kp, ifTi := LC601_PID_Ti, ifTd := LC601_PID_Td, ixManMode := LC601_MAN, ifManMv := LC601_PID_fMan);
LC601_OP := LC601_PID.qfMv;
(* Kjoele regulering *)
LC601_T(rIn := RT601_CS - RT601_CT, rOn := LC601_T_On, rOff := LC601_T_Off);
LC601_CMD := LC601_T.xOut;
END_FUNCTION_BLOCK

FUNCTION_BLOCK fbRomtype_11111112
  VAR_INPUT
    RB601_HVAC : BOOL;
    RT601_CT : REAL;
    RT601_SP_D : REAL;
    RT601_SP_S : REAL;
    RT601_SP_N : REAL;
    RT601_SP_F : REAL;
    OPM : INT;
    RY601_CV : REAL;
    RY601_SP : REAL;
    RY601_MAN : BOOL;
    LH601_MAN : BOOL;
    LC601_SP : REAL;
    LC601_MAN : BOOL;
  END_VAR
  VAR
    RY601_PID_Man : BOOL;  (* Co2 regulering *)
    RY601_PID_ManVal : REAL;
    RY601_PID : fbSE_PID;
    RY601_PID_Kp : REAL := 1;  (* PID Luft rom. Forsterkning *)
    RY601_PID_Ti : REAL := 10;  (* PID luft rom. I-tid *)
    RY601_PID_Td : REAL;  (* PID luft rom. D-tid *)
    RY601_PID_Zero : REAL;  (* PID luft rom. 0-punkt *)
    RY601_PID_Max : REAL := 2000;  (* PID luft rom. Max verdi ppm *)
    RY601_PID_fMan : REAL := 100;  (* PID varme rom. Manuelt kjoeling *)
    LH601_PID : fbSE_PID;  (* PID varme rom *)
    LH601_PID_Kp : REAL := 1;  (* PID varme rom. Forsterkning *)
    LH601_PID_Ti : REAL := 10;  (* PID varme rom. I-tid *)
    LH601_PID_Td : REAL;  (* PID varme rom. D-tid *)
    LH601_PID_fMan : REAL := 100;  (* PID varme rom. Manuelt paadrag *)
    LH601_T : fbSE_Hyst;  (* Termostat varme rom *)
    LH601_T_On : REAL := 0.5;
    LH601_T_Off : REAL := 0.1;
    LC601_PID : fbSE_PID;  (* PID kjoeling rom *)
    LC601_PID_Kp : REAL := 1;  (* PID kjoeling rom. Forsterkning *)
    LC601_PID_Ti : REAL := 10;  (* PID kjoeling rom. I-tid *)
    LC601_PID_Td : REAL;  (* PID kjoeling rom. D-tid *)
    LC601_PID_fMan : REAL := 100;  (* PID varme rom. Manuelt kjoeling *)
    LC601_T : fbSE_Hyst;  (* Termostat kjoeling rom *)
    LC601_T_On : REAL := 0.5;
    LC601_T_Off : REAL := 0.1;
  END_VAR
  VAR_OUTPUT
    OPM_CV : INT;
    RT601_CS : REAL;
    RY601_OP : REAL;
    LH601_OP : REAL;
    LH601_CMD : BOOL;
    LC601_OP : REAL;
    LC601_CMD : BOOL;
    LC602_CMD : BOOL;
  END_VAR

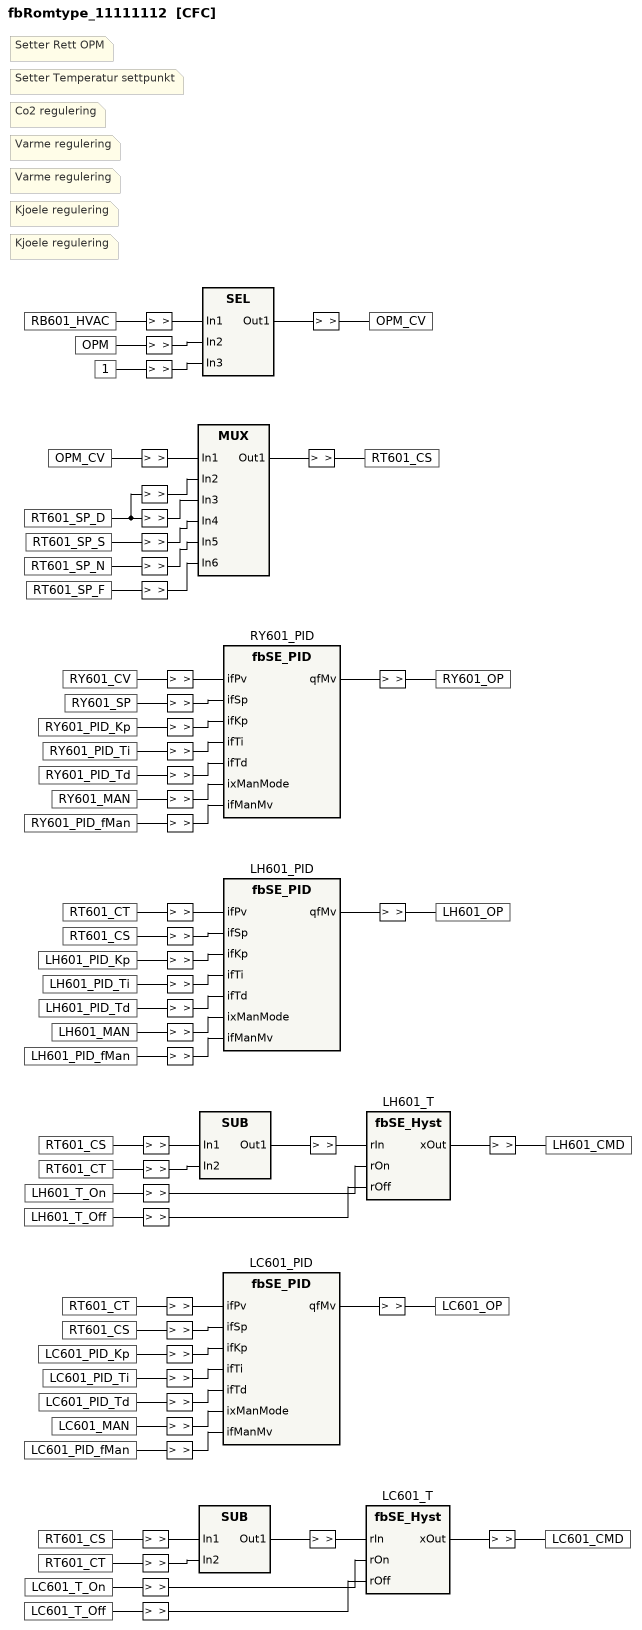
(* CFC diagram, written out as Structured Text *)
(* Setter Rett OPM *)
OPM_CV := SEL(RB601_HVAC, OPM, 1);
(* Setter Temperatur settpunkt *)
RT601_CS := MUX(OPM_CV, RT601_SP_D, RT601_SP_D, RT601_SP_S, RT601_SP_N, RT601_SP_F);
(* Co2 regulering *)
RY601_PID(ifPv := RY601_CV, ifSp := RY601_SP, ifKp := RY601_PID_Kp, ifTi := RY601_PID_Ti, ifTd := RY601_PID_Td, ixManMode := RY601_MAN, ifManMv := RY601_PID_fMan);
RY601_OP := RY601_PID.qfMv;
(* Varme regulering *)
LH601_PID(ifPv := RT601_CT, ifSp := RT601_CS, ifKp := LH601_PID_Kp, ifTi := LH601_PID_Ti, ifTd := LH601_PID_Td, ixManMode := LH601_MAN, ifManMv := LH601_PID_fMan);
LH601_OP := LH601_PID.qfMv;
(* Varme regulering *)
LH601_T(rIn := RT601_CS - RT601_CT, rOn := LH601_T_On, rOff := LH601_T_Off);
LH601_CMD := LH601_T.xOut;
(* Kjoele regulering *)
LC601_PID(ifPv := RT601_CT, ifSp := RT601_CS, ifKp := LC601_PID_Kp, ifTi := LC601_PID_Ti, ifTd := LC601_PID_Td, ixManMode := LC601_MAN, ifManMv := LC601_PID_fMan);
LC601_OP := LC601_PID.qfMv;
(* Kjoele regulering *)
LC601_T(rIn := RT601_CS - RT601_CT, rOn := LC601_T_On, rOff := LC601_T_Off);
LC601_CMD := LC601_T.xOut;
END_FUNCTION_BLOCK

FUNCTION_BLOCK fbRomtype_11212111
  VAR_INPUT
    RB601_HVAC : BOOL;
    RT601_CT : REAL;
    RT602_CT : REAL;
    RT600_SP_D : REAL;
    RT600_SP_S : REAL;
    RT600_SP_N : REAL;
    RT600_SP_F : REAL;
    OPM : INT;
    RY601_CV : REAL;
    RY601_SP : REAL;
    RY601_MAN : BOOL;
    LH600_MAN : BOOL;
    LC600_SP : REAL;
    LC600_MAN : BOOL;
  END_VAR
  VAR
    RY601_PID_Man : BOOL;  (* Co2 regulering *)
    RY601_PID_ManVal : REAL;
    RY601_PID : fbSE_PID;
    RY601_PID_Kp : REAL := 1;  (* PID Luft rom. Forsterkning *)
    RY601_PID_Ti : REAL := 10;  (* PID luft rom. I-tid *)
    RY601_PID_Td : REAL;  (* PID luft rom. D-tid *)
    RY601_PID_Zero : REAL;  (* PID luft rom. 0-punkt *)
    RY601_PID_Max : REAL := 2000;  (* PID luft rom. Max verdi ppm *)
    RY601_PID_fMan : REAL := 100;  (* PID varme rom. Manuelt kjoeling *)
    LH600_PID : fbSE_PID;  (* PID varme rom *)
    LH600_PID_Kp : REAL := 1;  (* PID varme rom. Forsterkning *)
    LH600_PID_Ti : REAL := 10;  (* PID varme rom. I-tid *)
    LH600_PID_Td : REAL;  (* PID varme rom. D-tid *)
    LH600_PID_fMan : REAL := 100;  (* PID varme rom. Manuelt paadrag *)
    LH600_T : fbSE_Hyst;  (* Termostat varme rom *)
    LH600_T_On : REAL := 0.5;
    LH600_T_Off : REAL := 0.1;
    LC600_PID : fbSE_PID;  (* PID kjoeling rom *)
    LC600_PID_Kp : REAL := 1;  (* PID kjoeling rom. Forsterkning *)
    LC600_PID_Ti : REAL := 10;  (* PID kjoeling rom. I-tid *)
    LC600_PID_Td : REAL;  (* PID kjoeling rom. D-tid *)
    LC600_PID_fMan : REAL := 100;  (* PID varme rom. Manuelt kjoeling *)
    LC600_T : fbSE_Hyst;  (* Termostat kjoeling rom *)
    LC600_T_On : REAL := 0.5;
    LC600_T_Off : REAL := 0.1;
  END_VAR
  VAR_OUTPUT
    OPM_CV : INT;
    RT600_CT : REAL;
    RT600_CS : REAL;
    RY601_OP : REAL;
    LH601_OP : REAL;
    LH602_OP : REAL;
    LH601_CMD : BOOL;
    LC601_OP : REAL;
    LC601_CMD : BOOL;
  END_VAR
  VAR  (* added by the conversion: wires and edge detectors of the diagram *)
    _ADD30_OUT : REAL;
    _DIV39_ENO : BOOL;
    _DIV39_OUT : REAL;
  END_VAR

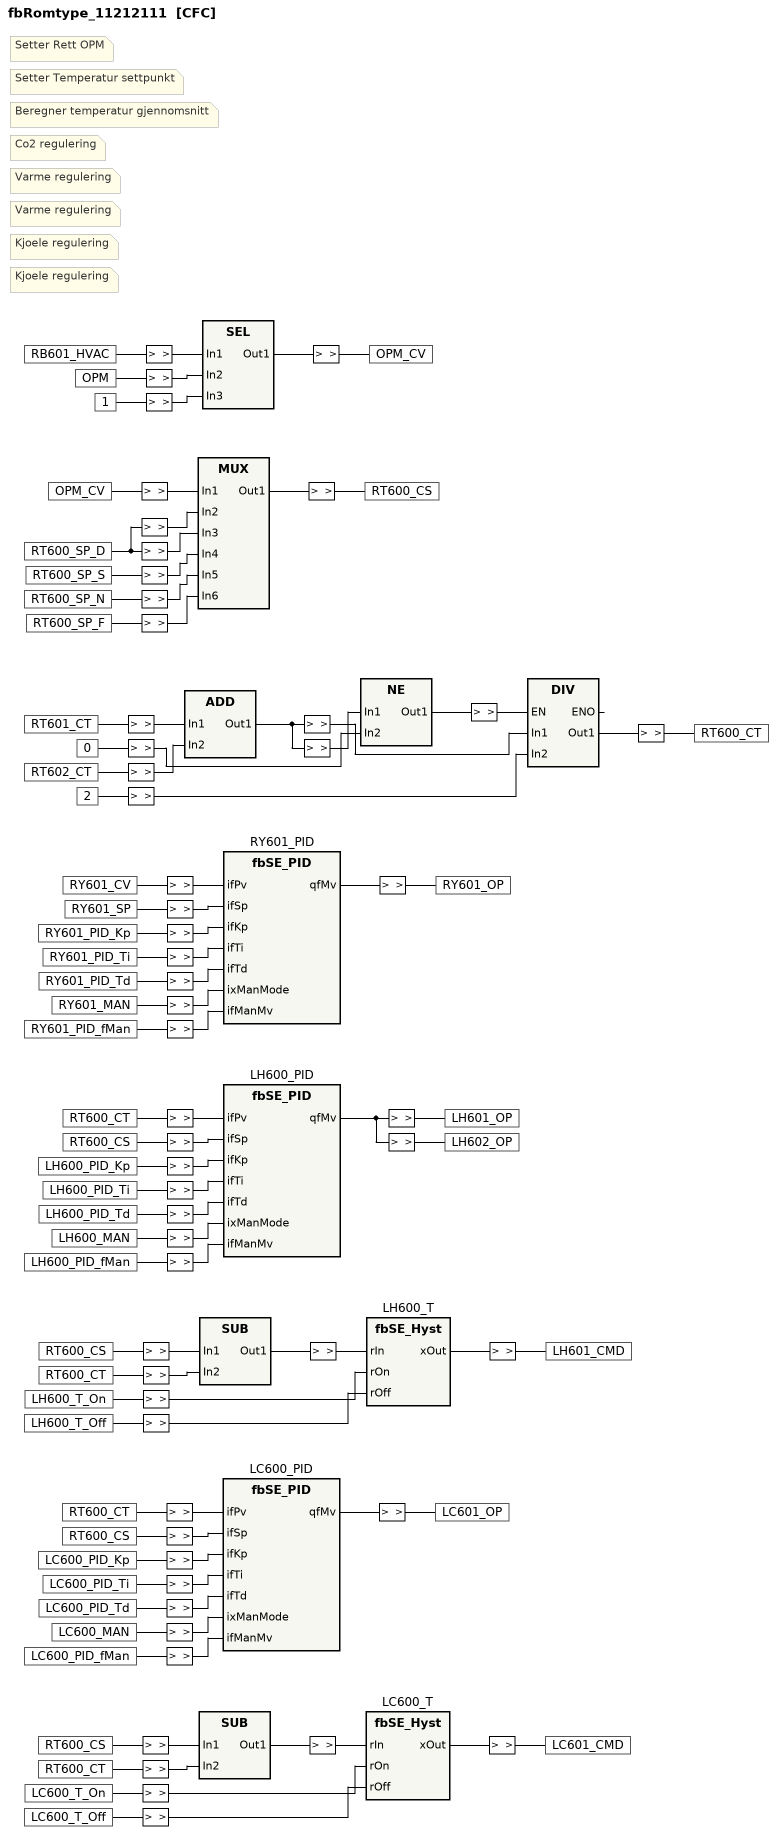
(* CFC diagram, written out as Structured Text *)
(* Setter Rett OPM *)
OPM_CV := SEL(RB601_HVAC, OPM, 1);
(* Setter Temperatur settpunkt *)
RT600_CS := MUX(OPM_CV, RT600_SP_D, RT600_SP_D, RT600_SP_S, RT600_SP_N, RT600_SP_F);
(* Beregner temperatur gjennomsnitt *)
_ADD30_OUT := RT601_CT + RT602_CT;
_DIV39_OUT := DIV(EN := _ADD30_OUT <> 0, IN1 := _ADD30_OUT, IN2 := 2, ENO => _DIV39_ENO);
IF _DIV39_ENO THEN RT600_CT := _DIV39_OUT; END_IF;
(* Co2 regulering *)
RY601_PID(ifPv := RY601_CV, ifSp := RY601_SP, ifKp := RY601_PID_Kp, ifTi := RY601_PID_Ti, ifTd := RY601_PID_Td, ixManMode := RY601_MAN, ifManMv := RY601_PID_fMan);
RY601_OP := RY601_PID.qfMv;
(* Varme regulering *)
LH600_PID(ifPv := RT600_CT, ifSp := RT600_CS, ifKp := LH600_PID_Kp, ifTi := LH600_PID_Ti, ifTd := LH600_PID_Td, ixManMode := LH600_MAN, ifManMv := LH600_PID_fMan);
LH601_OP := LH600_PID.qfMv;
LH602_OP := LH600_PID.qfMv;
(* Varme regulering *)
LH600_T(rIn := RT600_CS - RT600_CT, rOn := LH600_T_On, rOff := LH600_T_Off);
LH601_CMD := LH600_T.xOut;
(* Kjoele regulering *)
LC600_PID(ifPv := RT600_CT, ifSp := RT600_CS, ifKp := LC600_PID_Kp, ifTi := LC600_PID_Ti, ifTd := LC600_PID_Td, ixManMode := LC600_MAN, ifManMv := LC600_PID_fMan);
LC601_OP := LC600_PID.qfMv;
(* Kjoele regulering *)
LC600_T(rIn := RT600_CS - RT600_CT, rOn := LC600_T_On, rOff := LC600_T_Off);
LC601_CMD := LC600_T.xOut;
END_FUNCTION_BLOCK

FUNCTION_BLOCK fbRomtype_11211211
  VAR_INPUT
    RB601_HVAC : BOOL;
    RT601_CT : REAL;
    RT602_CT : REAL;
    RT600_SP_D : REAL;
    RT600_SP_S : REAL;
    RT600_SP_N : REAL;
    RT600_SP_F : REAL;
    OPM : INT;
    RY601_CV : REAL;
    RY601_SP : REAL;
    RY601_MAN : BOOL;
    LH600_MAN : BOOL;
    LC600_SP : REAL;
    LC600_MAN : BOOL;
  END_VAR
  VAR
    RY601_PID_Man : BOOL;  (* Co2 regulering *)
    RY601_PID_ManVal : REAL;
    RY601_PID : fbSE_PID;
    RY601_PID_Kp : REAL := 1;  (* PID Luft rom. Forsterkning *)
    RY601_PID_Ti : REAL := 10;  (* PID luft rom. I-tid *)
    RY601_PID_Td : REAL;  (* PID luft rom. D-tid *)
    RY601_PID_Zero : REAL;  (* PID luft rom. 0-punkt *)
    RY601_PID_Max : REAL := 2000;  (* PID luft rom. Max verdi ppm *)
    RY601_PID_fMan : REAL := 100;  (* PID varme rom. Manuelt kjoeling *)
    LH600_PID : fbSE_PID;  (* PID varme rom *)
    LH600_PID_Kp : REAL := 1;  (* PID varme rom. Forsterkning *)
    LH600_PID_Ti : REAL := 10;  (* PID varme rom. I-tid *)
    LH600_PID_Td : REAL;  (* PID varme rom. D-tid *)
    LH600_PID_fMan : REAL := 100;  (* PID varme rom. Manuelt paadrag *)
    LH600_T : fbSE_Hyst;  (* Termostat varme rom *)
    LH600_T_On : REAL := 0.5;
    LH600_T_Off : REAL := 0.1;
    LC600_PID : fbSE_PID;  (* PID kjoeling rom *)
    LC600_PID_Kp : REAL := 1;  (* PID kjoeling rom. Forsterkning *)
    LC600_PID_Ti : REAL := 10;  (* PID kjoeling rom. I-tid *)
    LC600_PID_Td : REAL;  (* PID kjoeling rom. D-tid *)
    LC600_PID_fMan : REAL := 100;  (* PID varme rom. Manuelt kjoeling *)
    LC600_T : fbSE_Hyst;  (* Termostat kjoeling rom *)
    LC600_T_On : REAL := 0.5;
    LC600_T_Off : REAL := 0.1;
  END_VAR
  VAR_OUTPUT
    OPM_CV : INT;
    RT600_CT : REAL;
    RT600_CS : REAL;
    RY601_OP : REAL;
    LH601_OP : REAL;
    LH601_CMD : BOOL;
    LH602_CMD : BOOL;
    LC601_OP : REAL;
    LC601_CMD : BOOL;
  END_VAR
  VAR  (* added by the conversion: wires and edge detectors of the diagram *)
    _ADD30_OUT : REAL;
    _DIV39_ENO : BOOL;
    _DIV39_OUT : REAL;
  END_VAR

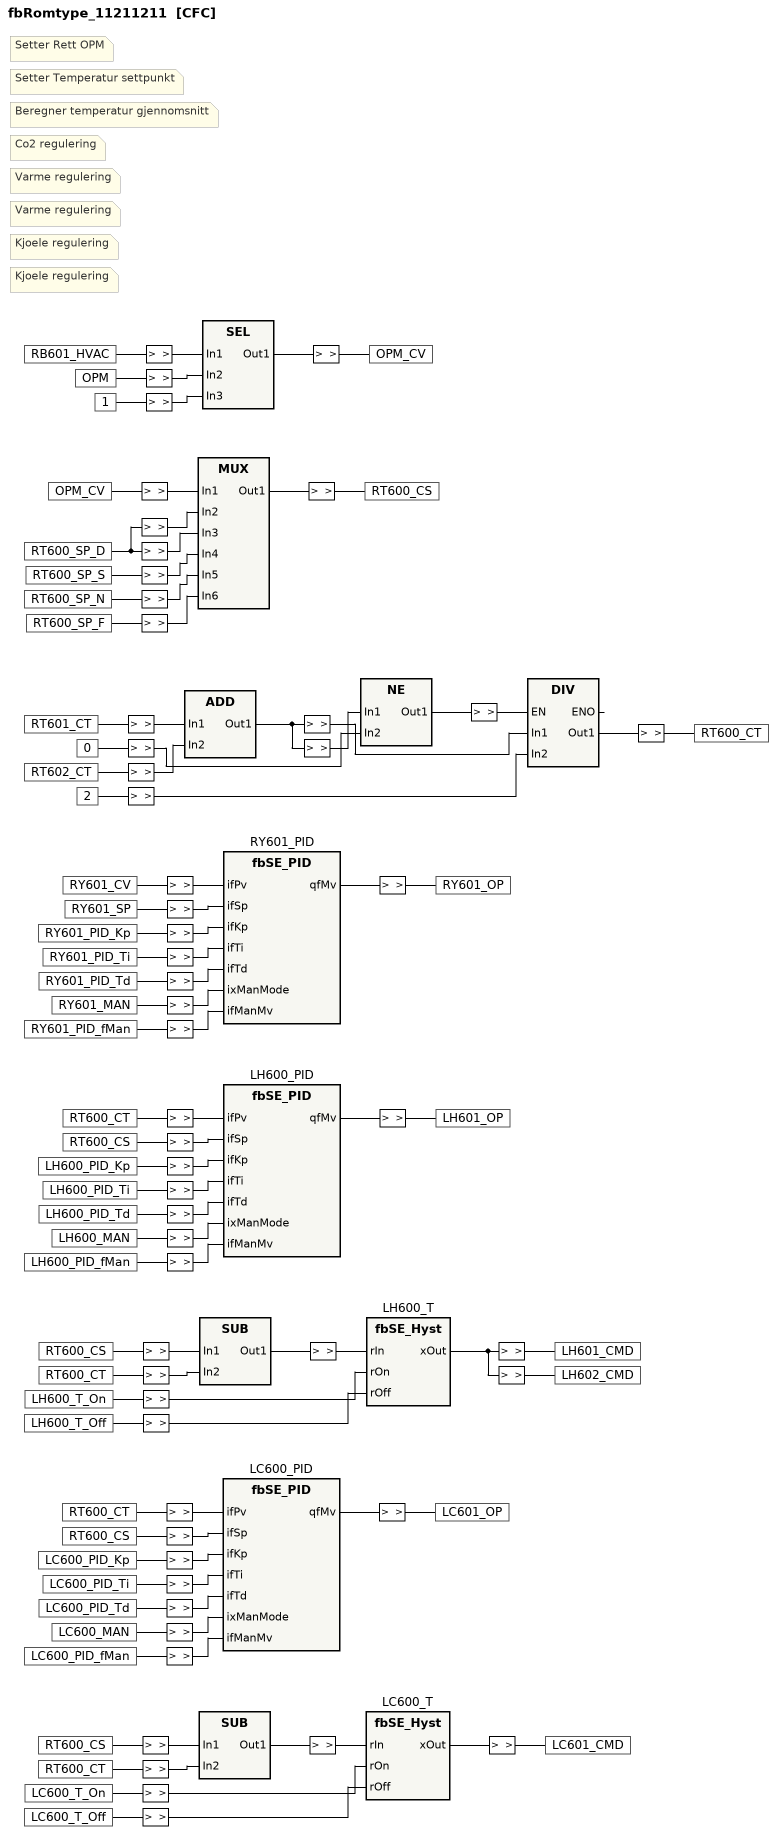
(* CFC diagram, written out as Structured Text *)
(* Setter Rett OPM *)
OPM_CV := SEL(RB601_HVAC, OPM, 1);
(* Setter Temperatur settpunkt *)
RT600_CS := MUX(OPM_CV, RT600_SP_D, RT600_SP_D, RT600_SP_S, RT600_SP_N, RT600_SP_F);
(* Beregner temperatur gjennomsnitt *)
_ADD30_OUT := RT601_CT + RT602_CT;
_DIV39_OUT := DIV(EN := _ADD30_OUT <> 0, IN1 := _ADD30_OUT, IN2 := 2, ENO => _DIV39_ENO);
IF _DIV39_ENO THEN RT600_CT := _DIV39_OUT; END_IF;
(* Co2 regulering *)
RY601_PID(ifPv := RY601_CV, ifSp := RY601_SP, ifKp := RY601_PID_Kp, ifTi := RY601_PID_Ti, ifTd := RY601_PID_Td, ixManMode := RY601_MAN, ifManMv := RY601_PID_fMan);
RY601_OP := RY601_PID.qfMv;
(* Varme regulering *)
LH600_PID(ifPv := RT600_CT, ifSp := RT600_CS, ifKp := LH600_PID_Kp, ifTi := LH600_PID_Ti, ifTd := LH600_PID_Td, ixManMode := LH600_MAN, ifManMv := LH600_PID_fMan);
LH601_OP := LH600_PID.qfMv;
(* Varme regulering *)
LH600_T(rIn := RT600_CS - RT600_CT, rOn := LH600_T_On, rOff := LH600_T_Off);
LH601_CMD := LH600_T.xOut;
LH602_CMD := LH600_T.xOut;
(* Kjoele regulering *)
LC600_PID(ifPv := RT600_CT, ifSp := RT600_CS, ifKp := LC600_PID_Kp, ifTi := LC600_PID_Ti, ifTd := LC600_PID_Td, ixManMode := LC600_MAN, ifManMv := LC600_PID_fMan);
LC601_OP := LC600_PID.qfMv;
(* Kjoele regulering *)
LC600_T(rIn := RT600_CS - RT600_CT, rOn := LC600_T_On, rOff := LC600_T_Off);
LC601_CMD := LC600_T.xOut;
END_FUNCTION_BLOCK

FUNCTION_BLOCK fbRomtype_11211121
  VAR_INPUT
    RB601_HVAC : BOOL;
    RT601_CT : REAL;
    RT602_CT : REAL;
    RT600_SP_D : REAL;
    RT600_SP_S : REAL;
    RT600_SP_N : REAL;
    RT600_SP_F : REAL;
    OPM : INT;
    RY601_CV : REAL;
    RY601_SP : REAL;
    RY601_MAN : BOOL;
    LH600_MAN : BOOL;
    LC600_SP : REAL;
    LC600_MAN : BOOL;
  END_VAR
  VAR
    RY601_PID_Man : BOOL;  (* Co2 regulering *)
    RY601_PID_ManVal : REAL;
    RY601_PID : fbSE_PID;
    RY601_PID_Kp : REAL := 1;  (* PID Luft rom. Forsterkning *)
    RY601_PID_Ti : REAL := 10;  (* PID luft rom. I-tid *)
    RY601_PID_Td : REAL;  (* PID luft rom. D-tid *)
    RY601_PID_Zero : REAL;  (* PID luft rom. 0-punkt *)
    RY601_PID_Max : REAL := 2000;  (* PID luft rom. Max verdi ppm *)
    RY601_PID_fMan : REAL := 100;  (* PID varme rom. Manuelt kjoeling *)
    LH600_PID : fbSE_PID;  (* PID varme rom *)
    LH600_PID_Kp : REAL := 1;  (* PID varme rom. Forsterkning *)
    LH600_PID_Ti : REAL := 10;  (* PID varme rom. I-tid *)
    LH600_PID_Td : REAL;  (* PID varme rom. D-tid *)
    LH600_PID_fMan : REAL := 100;  (* PID varme rom. Manuelt paadrag *)
    LH600_T : fbSE_Hyst;  (* Termostat varme rom *)
    LH600_T_On : REAL := 0.5;
    LH600_T_Off : REAL := 0.1;
    LC600_PID : fbSE_PID;  (* PID kjoeling rom *)
    LC600_PID_Kp : REAL := 1;  (* PID kjoeling rom. Forsterkning *)
    LC600_PID_Ti : REAL := 10;  (* PID kjoeling rom. I-tid *)
    LC600_PID_Td : REAL;  (* PID kjoeling rom. D-tid *)
    LC600_PID_fMan : REAL := 100;  (* PID varme rom. Manuelt kjoeling *)
    LC600_T : fbSE_Hyst;  (* Termostat kjoeling rom *)
    LC600_T_On : REAL := 0.5;
    LC600_T_Off : REAL := 0.1;
  END_VAR
  VAR_OUTPUT
    OPM_CV : INT;
    RT600_CT : REAL;
    RT600_CS : REAL;
    RY601_OP : REAL;
    LH601_OP : REAL;
    LH601_CMD : BOOL;
    LC601_OP : REAL;
    LC602_OP : REAL;
    LC601_CMD : BOOL;
  END_VAR
  VAR  (* added by the conversion: wires and edge detectors of the diagram *)
    _ADD30_OUT : REAL;
    _DIV39_ENO : BOOL;
    _DIV39_OUT : REAL;
  END_VAR

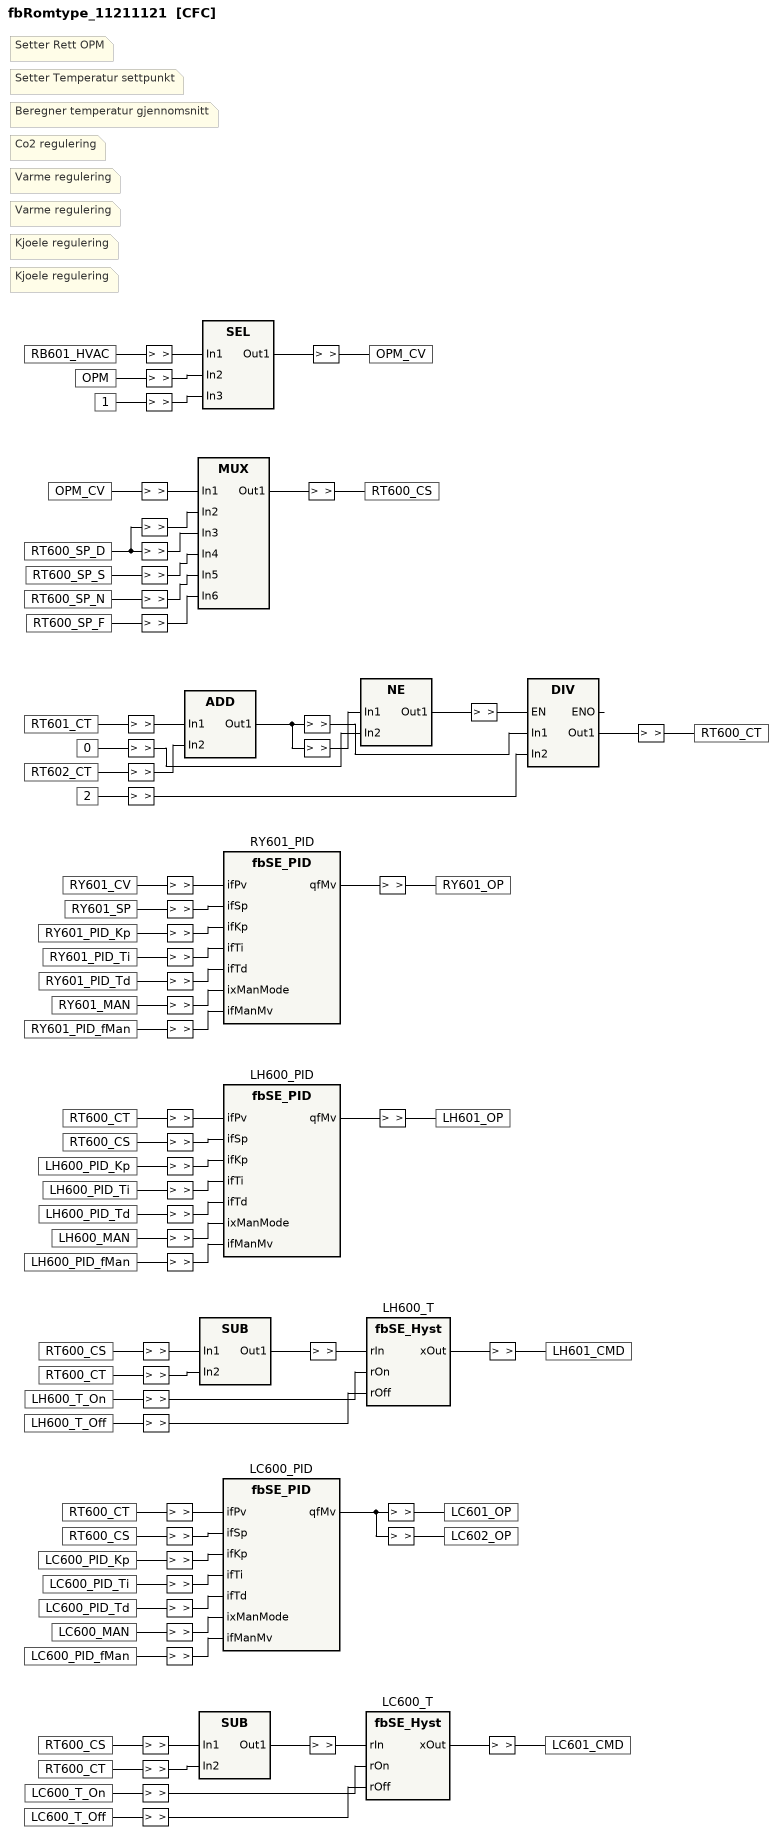
(* CFC diagram, written out as Structured Text *)
(* Setter Rett OPM *)
OPM_CV := SEL(RB601_HVAC, OPM, 1);
(* Setter Temperatur settpunkt *)
RT600_CS := MUX(OPM_CV, RT600_SP_D, RT600_SP_D, RT600_SP_S, RT600_SP_N, RT600_SP_F);
(* Beregner temperatur gjennomsnitt *)
_ADD30_OUT := RT601_CT + RT602_CT;
_DIV39_OUT := DIV(EN := _ADD30_OUT <> 0, IN1 := _ADD30_OUT, IN2 := 2, ENO => _DIV39_ENO);
IF _DIV39_ENO THEN RT600_CT := _DIV39_OUT; END_IF;
(* Co2 regulering *)
RY601_PID(ifPv := RY601_CV, ifSp := RY601_SP, ifKp := RY601_PID_Kp, ifTi := RY601_PID_Ti, ifTd := RY601_PID_Td, ixManMode := RY601_MAN, ifManMv := RY601_PID_fMan);
RY601_OP := RY601_PID.qfMv;
(* Varme regulering *)
LH600_PID(ifPv := RT600_CT, ifSp := RT600_CS, ifKp := LH600_PID_Kp, ifTi := LH600_PID_Ti, ifTd := LH600_PID_Td, ixManMode := LH600_MAN, ifManMv := LH600_PID_fMan);
LH601_OP := LH600_PID.qfMv;
(* Varme regulering *)
LH600_T(rIn := RT600_CS - RT600_CT, rOn := LH600_T_On, rOff := LH600_T_Off);
LH601_CMD := LH600_T.xOut;
(* Kjoele regulering *)
LC600_PID(ifPv := RT600_CT, ifSp := RT600_CS, ifKp := LC600_PID_Kp, ifTi := LC600_PID_Ti, ifTd := LC600_PID_Td, ixManMode := LC600_MAN, ifManMv := LC600_PID_fMan);
LC601_OP := LC600_PID.qfMv;
LC602_OP := LC600_PID.qfMv;
(* Kjoele regulering *)
LC600_T(rIn := RT600_CS - RT600_CT, rOn := LC600_T_On, rOff := LC600_T_Off);
LC601_CMD := LC600_T.xOut;
END_FUNCTION_BLOCK

FUNCTION_BLOCK fbRomtype_11211112
  VAR_INPUT
    RB601_HVAC : BOOL;
    RT601_CT : REAL;
    RT602_CT : REAL;
    RT600_SP_D : REAL;
    RT600_SP_S : REAL;
    RT600_SP_N : REAL;
    RT600_SP_F : REAL;
    OPM : INT;
    RY601_CV : REAL;
    RY601_SP : REAL;
    RY601_MAN : BOOL;
    LH600_MAN : BOOL;
    LC600_SP : REAL;
    LC600_MAN : BOOL;
  END_VAR
  VAR
    RY601_PID_Man : BOOL;  (* Co2 regulering *)
    RY601_PID_ManVal : REAL;
    RY601_PID : fbSE_PID;
    RY601_PID_Kp : REAL := 1;  (* PID Luft rom. Forsterkning *)
    RY601_PID_Ti : REAL := 10;  (* PID luft rom. I-tid *)
    RY601_PID_Td : REAL;  (* PID luft rom. D-tid *)
    RY601_PID_Zero : REAL;  (* PID luft rom. 0-punkt *)
    RY601_PID_Max : REAL := 2000;  (* PID luft rom. Max verdi ppm *)
    RY601_PID_fMan : REAL := 100;  (* PID varme rom. Manuelt kjoeling *)
    LH600_PID : fbSE_PID;  (* PID varme rom *)
    LH600_PID_Kp : REAL := 1;  (* PID varme rom. Forsterkning *)
    LH600_PID_Ti : REAL := 10;  (* PID varme rom. I-tid *)
    LH600_PID_Td : REAL;  (* PID varme rom. D-tid *)
    LH600_PID_fMan : REAL := 100;  (* PID varme rom. Manuelt paadrag *)
    LH600_T : fbSE_Hyst;  (* Termostat varme rom *)
    LH600_T_On : REAL := 0.5;
    LH600_T_Off : REAL := 0.1;
    LC600_PID : fbSE_PID;  (* PID kjoeling rom *)
    LC600_PID_Kp : REAL := 1;  (* PID kjoeling rom. Forsterkning *)
    LC600_PID_Ti : REAL := 10;  (* PID kjoeling rom. I-tid *)
    LC600_PID_Td : REAL;  (* PID kjoeling rom. D-tid *)
    LC600_PID_fMan : REAL := 100;  (* PID varme rom. Manuelt kjoeling *)
    LC600_T : fbSE_Hyst;  (* Termostat kjoeling rom *)
    LC600_T_On : REAL := 0.5;
    LC600_T_Off : REAL := 0.1;
  END_VAR
  VAR_OUTPUT
    OPM_CV : INT;
    RT600_CT : REAL;
    RT600_CS : REAL;
    RY601_OP : REAL;
    LH601_OP : REAL;
    LH601_CMD : BOOL;
    LC601_OP : REAL;
    LC601_CMD : BOOL;
    LC602_CMD : BOOL;
  END_VAR
  VAR  (* added by the conversion: wires and edge detectors of the diagram *)
    _ADD30_OUT : REAL;
    _DIV39_ENO : BOOL;
    _DIV39_OUT : REAL;
  END_VAR

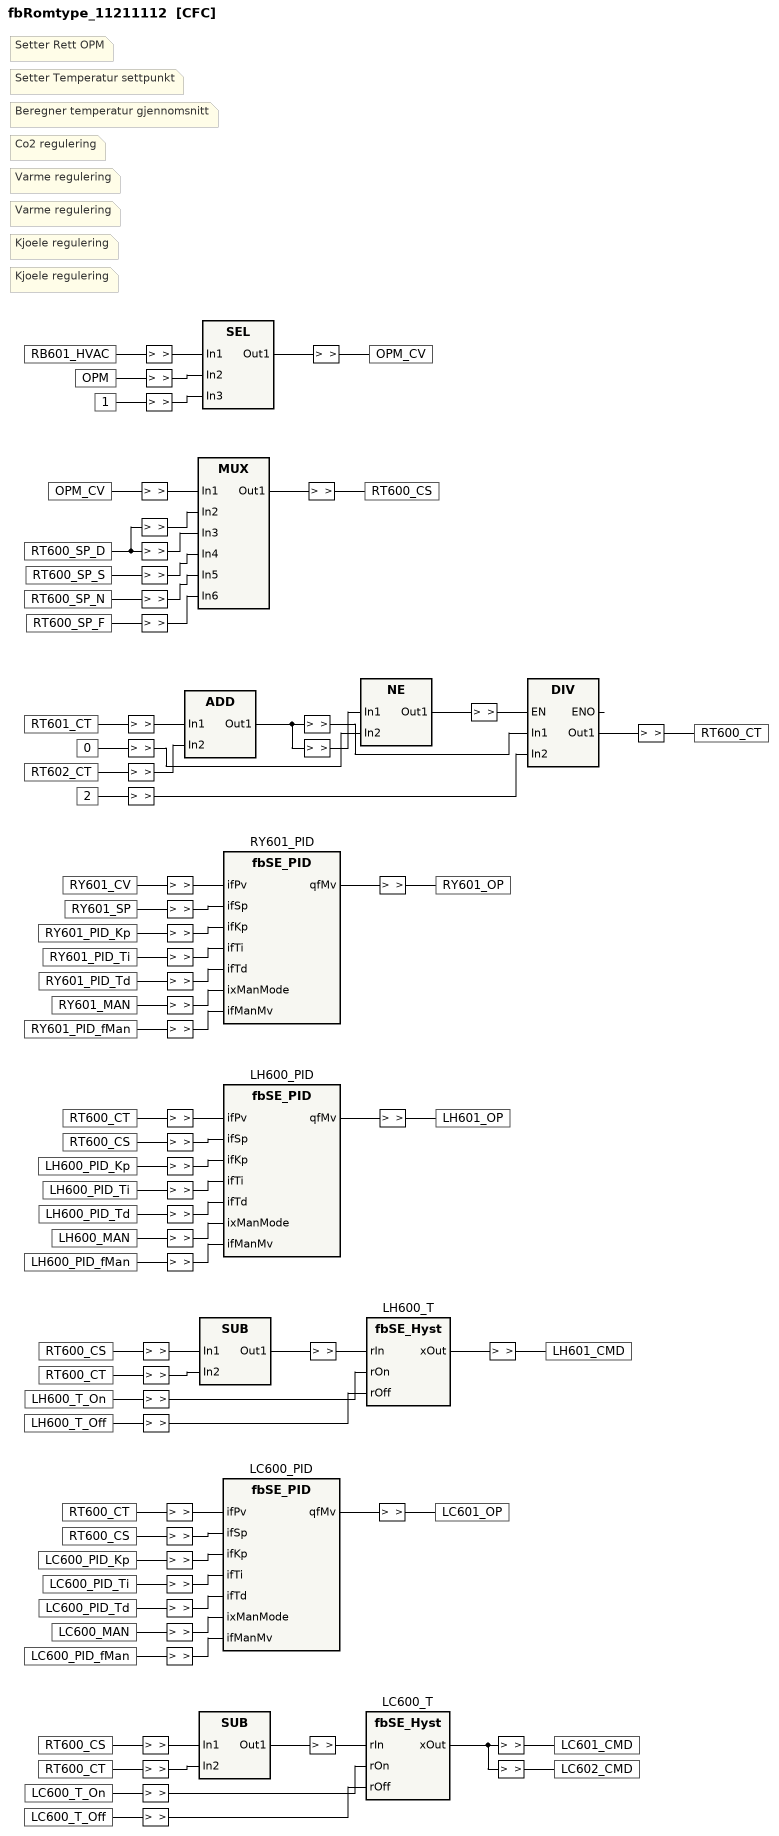
(* CFC diagram, written out as Structured Text *)
(* Setter Rett OPM *)
OPM_CV := SEL(RB601_HVAC, OPM, 1);
(* Setter Temperatur settpunkt *)
RT600_CS := MUX(OPM_CV, RT600_SP_D, RT600_SP_D, RT600_SP_S, RT600_SP_N, RT600_SP_F);
(* Beregner temperatur gjennomsnitt *)
_ADD30_OUT := RT601_CT + RT602_CT;
_DIV39_OUT := DIV(EN := _ADD30_OUT <> 0, IN1 := _ADD30_OUT, IN2 := 2, ENO => _DIV39_ENO);
IF _DIV39_ENO THEN RT600_CT := _DIV39_OUT; END_IF;
(* Co2 regulering *)
RY601_PID(ifPv := RY601_CV, ifSp := RY601_SP, ifKp := RY601_PID_Kp, ifTi := RY601_PID_Ti, ifTd := RY601_PID_Td, ixManMode := RY601_MAN, ifManMv := RY601_PID_fMan);
RY601_OP := RY601_PID.qfMv;
(* Varme regulering *)
LH600_PID(ifPv := RT600_CT, ifSp := RT600_CS, ifKp := LH600_PID_Kp, ifTi := LH600_PID_Ti, ifTd := LH600_PID_Td, ixManMode := LH600_MAN, ifManMv := LH600_PID_fMan);
LH601_OP := LH600_PID.qfMv;
(* Varme regulering *)
LH600_T(rIn := RT600_CS - RT600_CT, rOn := LH600_T_On, rOff := LH600_T_Off);
LH601_CMD := LH600_T.xOut;
(* Kjoele regulering *)
LC600_PID(ifPv := RT600_CT, ifSp := RT600_CS, ifKp := LC600_PID_Kp, ifTi := LC600_PID_Ti, ifTd := LC600_PID_Td, ixManMode := LC600_MAN, ifManMv := LC600_PID_fMan);
LC601_OP := LC600_PID.qfMv;
(* Kjoele regulering *)
LC600_T(rIn := RT600_CS - RT600_CT, rOn := LC600_T_On, rOff := LC600_T_Off);
LC601_CMD := LC600_T.xOut;
LC602_CMD := LC600_T.xOut;
END_FUNCTION_BLOCK

FUNCTION_BLOCK fbRomtype_11221111
  VAR_INPUT
    RB601_HVAC : BOOL;
    RT601_CT : REAL;
    RT602_CT : REAL;
    RT600_SP_D : REAL;
    RT600_SP_S : REAL;
    RT600_SP_N : REAL;
    RT600_SP_F : REAL;
    OPM : INT;
    RY601_CV : REAL;
    RY602_CV : REAL;
    RY600_SP : REAL;
    RY600_MAN : BOOL;
    LH600_MAN : BOOL;
    LC600_SP : REAL;
    LC600_MAN : BOOL;
  END_VAR
  VAR
    RY600_PID_Man : BOOL;  (* Co2 regulering *)
    RY600_PID_ManVal : REAL;
    RY600_PID : fbSE_PID;
    RY600_PID_Kp : REAL := 1;  (* PID Luft rom. Forsterkning *)
    RY600_PID_Ti : REAL := 10;  (* PID luft rom. I-tid *)
    RY600_PID_Td : REAL;  (* PID luft rom. D-tid *)
    RY600_PID_Zero : REAL;  (* PID luft rom. 0-punkt *)
    RY600_PID_Max : REAL := 2000;  (* PID luft rom. Max verdi ppm *)
    RY600_PID_fMan : REAL := 100;  (* PID varme rom. Manuelt kjoeling *)
    LH600_PID : fbSE_PID;  (* PID varme rom *)
    LH600_PID_Kp : REAL := 1;  (* PID varme rom. Forsterkning *)
    LH600_PID_Ti : REAL := 10;  (* PID varme rom. I-tid *)
    LH600_PID_Td : REAL;  (* PID varme rom. D-tid *)
    LH600_PID_fMan : REAL := 100;  (* PID varme rom. Manuelt paadrag *)
    LH600_T : fbSE_Hyst;  (* Termostat varme rom *)
    LH600_T_On : REAL := 0.5;
    LH600_T_Off : REAL := 0.1;
    LC600_PID : fbSE_PID;  (* PID kjoeling rom *)
    LC600_PID_Kp : REAL := 1;  (* PID kjoeling rom. Forsterkning *)
    LC600_PID_Ti : REAL := 10;  (* PID kjoeling rom. I-tid *)
    LC600_PID_Td : REAL;  (* PID kjoeling rom. D-tid *)
    LC600_PID_fMan : REAL := 100;  (* PID varme rom. Manuelt kjoeling *)
    LC600_T : fbSE_Hyst;  (* Termostat kjoeling rom *)
    LC600_T_On : REAL := 0.5;
    LC600_T_Off : REAL := 0.1;
  END_VAR
  VAR_OUTPUT
    OPM_CV : INT;
    RT600_CT : REAL;
    RT600_CS : REAL;
    RY600_CV : REAL;
    RY600_OP : REAL;
    LH601_OP : REAL;
    LH601_CMD : BOOL;
    LC601_OP : REAL;
    LC601_CMD : BOOL;
  END_VAR
  VAR  (* added by the conversion: wires and edge detectors of the diagram *)
    _ADD30_OUT : REAL;
    _DIV39_ENO : BOOL;
    _DIV39_OUT : REAL;
    _ADD49_OUT : REAL;
    _DIV58_ENO : BOOL;
    _DIV58_OUT : REAL;
  END_VAR

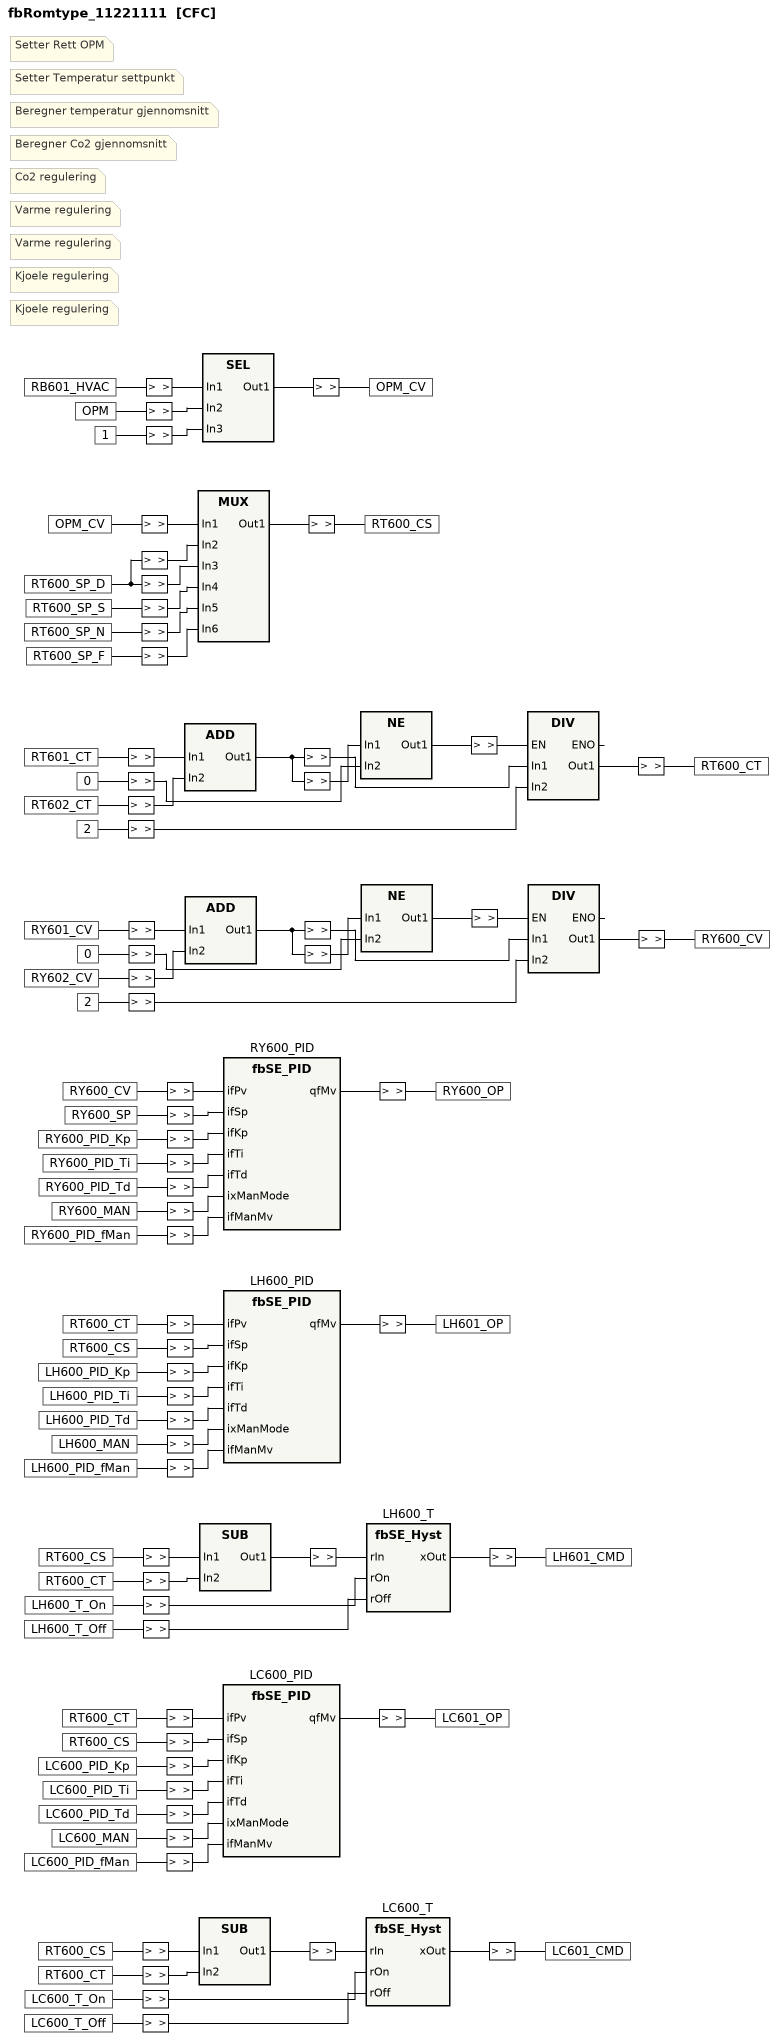
(* CFC diagram, written out as Structured Text *)
(* Setter Rett OPM *)
OPM_CV := SEL(RB601_HVAC, OPM, 1);
(* Setter Temperatur settpunkt *)
RT600_CS := MUX(OPM_CV, RT600_SP_D, RT600_SP_D, RT600_SP_S, RT600_SP_N, RT600_SP_F);
(* Beregner temperatur gjennomsnitt *)
_ADD30_OUT := RT601_CT + RT602_CT;
_DIV39_OUT := DIV(EN := _ADD30_OUT <> 0, IN1 := _ADD30_OUT, IN2 := 2, ENO => _DIV39_ENO);
IF _DIV39_ENO THEN RT600_CT := _DIV39_OUT; END_IF;
(* Beregner Co2 gjennomsnitt *)
_ADD49_OUT := RY601_CV + RY602_CV;
_DIV58_OUT := DIV(EN := _ADD49_OUT <> 0, IN1 := _ADD49_OUT, IN2 := 2, ENO => _DIV58_ENO);
IF _DIV58_ENO THEN RY600_CV := _DIV58_OUT; END_IF;
(* Co2 regulering *)
RY600_PID(ifPv := RY600_CV, ifSp := RY600_SP, ifKp := RY600_PID_Kp, ifTi := RY600_PID_Ti, ifTd := RY600_PID_Td, ixManMode := RY600_MAN, ifManMv := RY600_PID_fMan);
RY600_OP := RY600_PID.qfMv;
(* Varme regulering *)
LH600_PID(ifPv := RT600_CT, ifSp := RT600_CS, ifKp := LH600_PID_Kp, ifTi := LH600_PID_Ti, ifTd := LH600_PID_Td, ixManMode := LH600_MAN, ifManMv := LH600_PID_fMan);
LH601_OP := LH600_PID.qfMv;
(* Varme regulering *)
LH600_T(rIn := RT600_CS - RT600_CT, rOn := LH600_T_On, rOff := LH600_T_Off);
LH601_CMD := LH600_T.xOut;
(* Kjoele regulering *)
LC600_PID(ifPv := RT600_CT, ifSp := RT600_CS, ifKp := LC600_PID_Kp, ifTi := LC600_PID_Ti, ifTd := LC600_PID_Td, ixManMode := LC600_MAN, ifManMv := LC600_PID_fMan);
LC601_OP := LC600_PID.qfMv;
(* Kjoele regulering *)
LC600_T(rIn := RT600_CS - RT600_CT, rOn := LC600_T_On, rOff := LC600_T_Off);
LC601_CMD := LC600_T.xOut;
END_FUNCTION_BLOCK

FUNCTION_BLOCK fbRomtype_11222222
  VAR_INPUT
    RB601_HVAC : BOOL;
    RT601_CT : REAL;
    RT602_CT : REAL;
    RT600_SP_D : REAL;
    RT600_SP_S : REAL;
    RT600_SP_N : REAL;
    RT600_SP_F : REAL;
    OPM : INT;
    RY601_CV : REAL;
    RY602_CV : REAL;
    RY600_SP : REAL;
    RY600_MAN : BOOL;
    LH600_MAN : BOOL;
    LC600_SP : REAL;
    LC600_MAN : BOOL;
  END_VAR
  VAR
    RY600_PID_Man : BOOL;  (* Co2 regulering *)
    RY600_PID_ManVal : REAL;
    RY600_PID : fbSE_PID;
    RY600_PID_Kp : REAL := 1;  (* PID Luft rom. Forsterkning *)
    RY600_PID_Ti : REAL := 10;  (* PID luft rom. I-tid *)
    RY600_PID_Td : REAL;  (* PID luft rom. D-tid *)
    RY600_PID_Zero : REAL;  (* PID luft rom. 0-punkt *)
    RY600_PID_Max : REAL := 2000;  (* PID luft rom. Max verdi ppm *)
    RY600_PID_fMan : REAL := 100;  (* PID varme rom. Manuelt kjoeling *)
    LH600_PID : fbSE_PID;  (* PID varme rom *)
    LH600_PID_Kp : REAL := 1;  (* PID varme rom. Forsterkning *)
    LH600_PID_Ti : REAL := 10;  (* PID varme rom. I-tid *)
    LH600_PID_Td : REAL;  (* PID varme rom. D-tid *)
    LH600_PID_fMan : REAL := 100;  (* PID varme rom. Manuelt paadrag *)
    LH600_T : fbSE_Hyst;  (* Termostat varme rom *)
    LH600_T_On : REAL := 0.5;
    LH600_T_Off : REAL := 0.1;
    LC600_PID : fbSE_PID;  (* PID kjoeling rom *)
    LC600_PID_Kp : REAL := 1;  (* PID kjoeling rom. Forsterkning *)
    LC600_PID_Ti : REAL := 10;  (* PID kjoeling rom. I-tid *)
    LC600_PID_Td : REAL;  (* PID kjoeling rom. D-tid *)
    LC600_PID_fMan : REAL := 100;  (* PID varme rom. Manuelt kjoeling *)
    LC600_T : fbSE_Hyst;  (* Termostat kjoeling rom *)
    LC600_T_On : REAL := 0.5;
    LC600_T_Off : REAL := 0.1;
  END_VAR
  VAR_OUTPUT
    OPM_CV : INT;
    RT600_CT : REAL;
    RT600_CS : REAL;
    RY600_CV : REAL;
    RY600_OP : REAL;
    LH601_OP : REAL;
    LH602_OP : REAL;
    LH601_CMD : BOOL;
    LH602_CMD : BOOL;
    LC601_OP : REAL;
    LC602_OP : REAL;
    LC601_CMD : BOOL;
    LC602_CMD : BOOL;
  END_VAR
  VAR  (* added by the conversion: wires and edge detectors of the diagram *)
    _ADD30_OUT : REAL;
    _DIV39_ENO : BOOL;
    _DIV39_OUT : REAL;
    _ADD49_OUT : REAL;
    _DIV58_ENO : BOOL;
    _DIV58_OUT : REAL;
  END_VAR

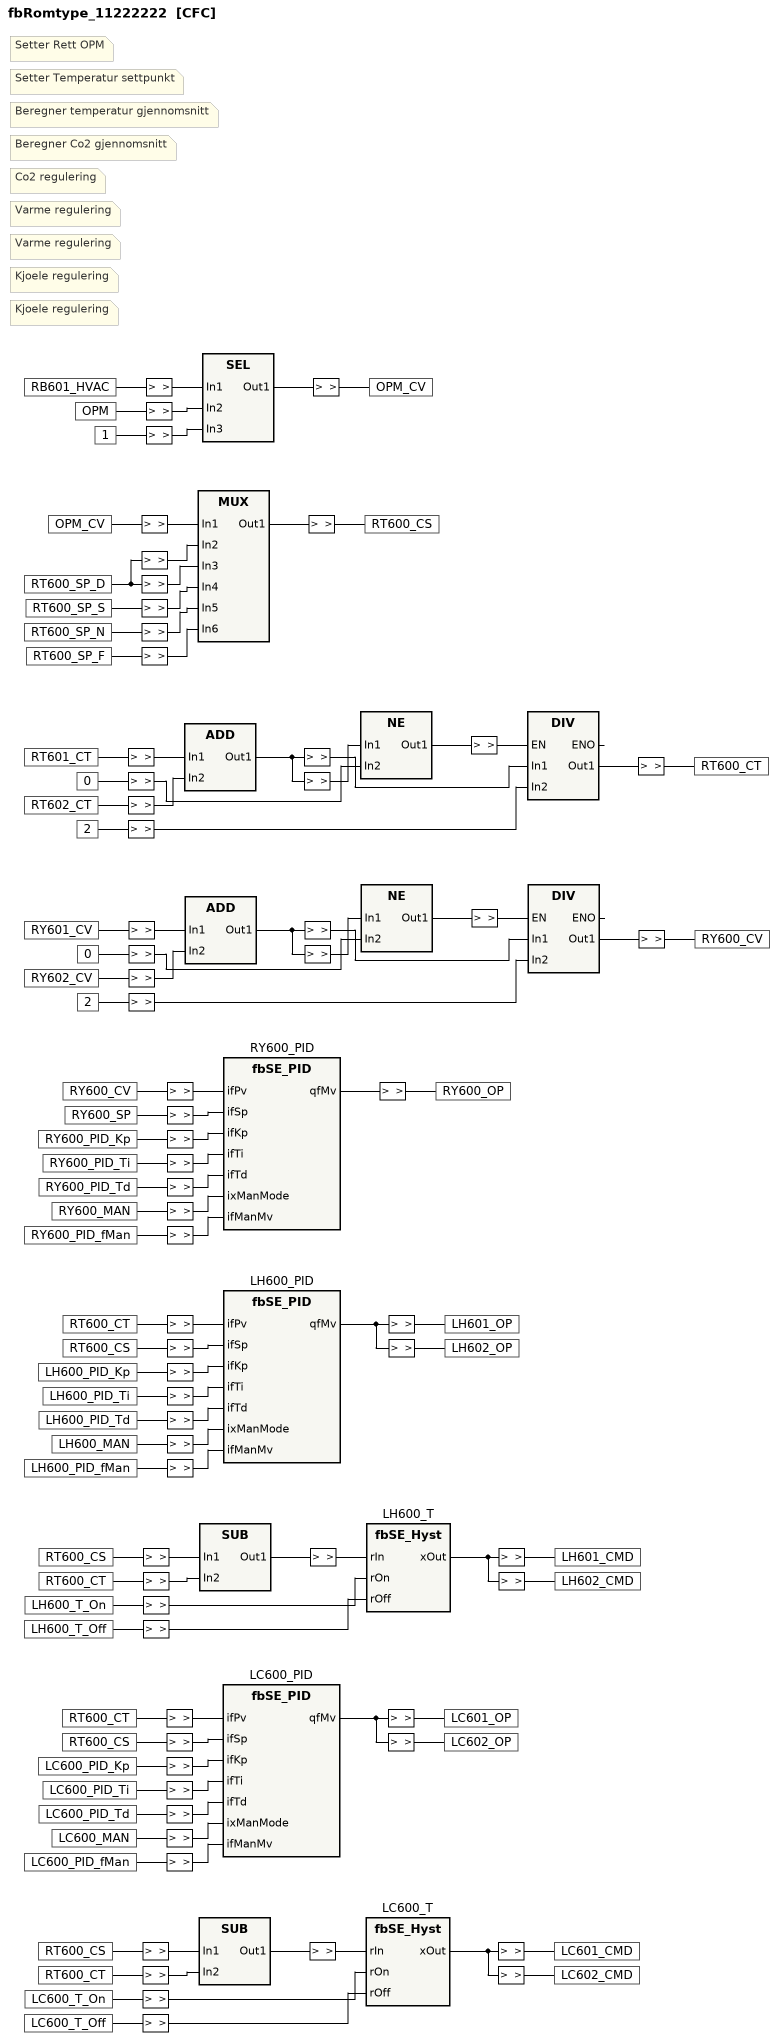
(* CFC diagram, written out as Structured Text *)
(* Setter Rett OPM *)
OPM_CV := SEL(RB601_HVAC, OPM, 1);
(* Setter Temperatur settpunkt *)
RT600_CS := MUX(OPM_CV, RT600_SP_D, RT600_SP_D, RT600_SP_S, RT600_SP_N, RT600_SP_F);
(* Beregner temperatur gjennomsnitt *)
_ADD30_OUT := RT601_CT + RT602_CT;
_DIV39_OUT := DIV(EN := _ADD30_OUT <> 0, IN1 := _ADD30_OUT, IN2 := 2, ENO => _DIV39_ENO);
IF _DIV39_ENO THEN RT600_CT := _DIV39_OUT; END_IF;
(* Beregner Co2 gjennomsnitt *)
_ADD49_OUT := RY601_CV + RY602_CV;
_DIV58_OUT := DIV(EN := _ADD49_OUT <> 0, IN1 := _ADD49_OUT, IN2 := 2, ENO => _DIV58_ENO);
IF _DIV58_ENO THEN RY600_CV := _DIV58_OUT; END_IF;
(* Co2 regulering *)
RY600_PID(ifPv := RY600_CV, ifSp := RY600_SP, ifKp := RY600_PID_Kp, ifTi := RY600_PID_Ti, ifTd := RY600_PID_Td, ixManMode := RY600_MAN, ifManMv := RY600_PID_fMan);
RY600_OP := RY600_PID.qfMv;
(* Varme regulering *)
LH600_PID(ifPv := RT600_CT, ifSp := RT600_CS, ifKp := LH600_PID_Kp, ifTi := LH600_PID_Ti, ifTd := LH600_PID_Td, ixManMode := LH600_MAN, ifManMv := LH600_PID_fMan);
LH601_OP := LH600_PID.qfMv;
LH602_OP := LH600_PID.qfMv;
(* Varme regulering *)
LH600_T(rIn := RT600_CS - RT600_CT, rOn := LH600_T_On, rOff := LH600_T_Off);
LH601_CMD := LH600_T.xOut;
LH602_CMD := LH600_T.xOut;
(* Kjoele regulering *)
LC600_PID(ifPv := RT600_CT, ifSp := RT600_CS, ifKp := LC600_PID_Kp, ifTi := LC600_PID_Ti, ifTd := LC600_PID_Td, ixManMode := LC600_MAN, ifManMv := LC600_PID_fMan);
LC601_OP := LC600_PID.qfMv;
LC602_OP := LC600_PID.qfMv;
(* Kjoele regulering *)
LC600_T(rIn := RT600_CS - RT600_CT, rOn := LC600_T_On, rOff := LC600_T_Off);
LC601_CMD := LC600_T.xOut;
LC602_CMD := LC600_T.xOut;
END_FUNCTION_BLOCK

FUNCTION_BLOCK fbRomtype_22222222
  VAR_INPUT
    RB601_HVAC : BOOL;
    RB602_HVAC : BOOL;
    RT601_CT : REAL;
    RT602_CT : REAL;
    RT600_SP_D : REAL;
    RT600_SP_S : REAL;
    RT600_SP_N : REAL;
    RT600_SP_F : REAL;
    OPM : INT;
    RY601_CV : REAL;
    RY602_CV : REAL;
    RY600_SP : REAL;
    RY600_MAN : BOOL;
    LH600_MAN : BOOL;
    LC600_SP : REAL;
    LC600_MAN : BOOL;
  END_VAR
  VAR
    RY600_PID_Man : BOOL;  (* Co2 regulering *)
    RY600_PID_ManVal : REAL;
    RY600_PID : fbSE_PID;
    RY600_PID_Kp : REAL := 1;  (* PID Luft rom. Forsterkning *)
    RY600_PID_Ti : REAL := 10;  (* PID luft rom. I-tid *)
    RY600_PID_Td : REAL;  (* PID luft rom. D-tid *)
    RY600_PID_Zero : REAL;  (* PID luft rom. 0-punkt *)
    RY600_PID_Max : REAL := 2000;  (* PID luft rom. Max verdi ppm *)
    RY600_PID_fMan : REAL := 100;  (* PID varme rom. Manuelt kjoeling *)
    LH600_PID : fbSE_PID;  (* PID varme rom *)
    LH600_PID_Kp : REAL := 1;  (* PID varme rom. Forsterkning *)
    LH600_PID_Ti : REAL := 10;  (* PID varme rom. I-tid *)
    LH600_PID_Td : REAL;  (* PID varme rom. D-tid *)
    LH600_PID_fMan : REAL := 100;  (* PID varme rom. Manuelt paadrag *)
    LH600_T : fbSE_Hyst;  (* Termostat varme rom *)
    LH600_T_On : REAL := 0.5;
    LH600_T_Off : REAL := 0.1;
    LC600_PID : fbSE_PID;  (* PID kjoeling rom *)
    LC600_PID_Kp : REAL := 1;  (* PID kjoeling rom. Forsterkning *)
    LC600_PID_Ti : REAL := 10;  (* PID kjoeling rom. I-tid *)
    LC600_PID_Td : REAL;  (* PID kjoeling rom. D-tid *)
    LC600_PID_fMan : REAL := 100;  (* PID varme rom. Manuelt kjoeling *)
    LC600_T : fbSE_Hyst;  (* Termostat kjoeling rom *)
    LC600_T_On : REAL := 0.5;
    LC600_T_Off : REAL := 0.1;
  END_VAR
  VAR_OUTPUT
    RB600_HVAC : BOOL;
    OPM_CV : INT;
    RT600_CT : REAL;
    RT600_CS : REAL;
    RY600_CV : REAL;
    RY600_OP : REAL;
    LH601_OP : REAL;
    LH602_OP : REAL;
    LH601_CMD : BOOL;
    LH602_CMD : BOOL;
    LC601_OP : REAL;
    LC602_OP : REAL;
    LC601_CMD : BOOL;
    LC602_CMD : BOOL;
  END_VAR
  VAR  (* added by the conversion: wires and edge detectors of the diagram *)
    _OR5_OUT : BOOL;
    _ADD36_OUT : REAL;
    _DIV45_ENO : BOOL;
    _DIV45_OUT : REAL;
    _ADD55_OUT : REAL;
    _DIV64_ENO : BOOL;
    _DIV64_OUT : REAL;
  END_VAR

(* CFC diagram, written out as Structured Text *)
(* Setter Rett OPM *)
_OR5_OUT := RB601_HVAC OR RB602_HVAC;
OPM_CV := SEL(_OR5_OUT, OPM, 1);
RB600_HVAC := _OR5_OUT;
(* Setter Temperatur settpunkt *)
RT600_CS := MUX(OPM_CV, RT600_SP_D, RT600_SP_D, RT600_SP_S, RT600_SP_N, RT600_SP_F);
(* Beregner temperatur gjennomsnitt *)
_ADD36_OUT := RT601_CT + RT602_CT;
_DIV45_OUT := DIV(EN := _ADD36_OUT <> 0, IN1 := _ADD36_OUT, IN2 := 2, ENO => _DIV45_ENO);
IF _DIV45_ENO THEN RT600_CT := _DIV45_OUT; END_IF;
(* Beregner Co2 gjennomsnitt *)
_ADD55_OUT := RY601_CV + RY602_CV;
_DIV64_OUT := DIV(EN := _ADD55_OUT <> 0, IN1 := _ADD55_OUT, IN2 := 2, ENO => _DIV64_ENO);
IF _DIV64_ENO THEN RY600_CV := _DIV64_OUT; END_IF;
(* Co2 regulering *)
RY600_PID(ifPv := RY600_CV, ifSp := RY600_SP, ifKp := RY600_PID_Kp, ifTi := RY600_PID_Ti, ifTd := RY600_PID_Td, ixManMode := RY600_MAN, ifManMv := RY600_PID_fMan);
RY600_OP := RY600_PID.qfMv;
(* Varme regulering *)
LH600_PID(ifPv := RT600_CT, ifSp := RT600_CS, ifKp := LH600_PID_Kp, ifTi := LH600_PID_Ti, ifTd := LH600_PID_Td, ixManMode := LH600_MAN, ifManMv := LH600_PID_fMan);
LH601_OP := LH600_PID.qfMv;
LH602_OP := LH600_PID.qfMv;
(* Varme regulering *)
LH600_T(rIn := RT600_CS - RT600_CT, rOn := LH600_T_On, rOff := LH600_T_Off);
LH601_CMD := LH600_T.xOut;
LH602_CMD := LH600_T.xOut;
(* Kjoele regulering *)
LC600_PID(ifPv := RT600_CT, ifSp := RT600_CS, ifKp := LC600_PID_Kp, ifTi := LC600_PID_Ti, ifTd := LC600_PID_Td, ixManMode := LC600_MAN, ifManMv := LC600_PID_fMan);
LC601_OP := LC600_PID.qfMv;
LC602_OP := LC600_PID.qfMv;
(* Kjoele regulering *)
LC600_T(rIn := RT600_CS - RT600_CT, rOn := LC600_T_On, rOff := LC600_T_Off);
LC601_CMD := LC600_T.xOut;
LC602_CMD := LC600_T.xOut;
END_FUNCTION_BLOCK

FUNCTION_BLOCK fbRomtype_22022222
  VAR_INPUT
    RB601_HVAC : BOOL;
    RB602_HVAC : BOOL;
    RY601_CV : REAL;
    RY602_CV : REAL;
    RY600_SP : REAL;
    RY600_MAN : BOOL;
    LH601_MAN : BOOL;
    LC601_SP : REAL;
    LC601_MAN : BOOL;
  END_VAR
  VAR
    RY600_PID_Man : BOOL;  (* Co2 regulering *)
    RY600_PID_ManVal : REAL;
    RY600_PID : fbSE_PID;
    RY600_PID_Kp : REAL := 1;  (* PID Luft rom. Forsterkning *)
    RY600_PID_Ti : REAL := 10;  (* PID luft rom. I-tid *)
    RY600_PID_Td : REAL;  (* PID luft rom. D-tid *)
    RY600_PID_Zero : REAL;  (* PID luft rom. 0-punkt *)
    RY600_PID_Max : REAL := 2000;  (* PID luft rom. Max verdi ppm *)
    RY600_PID_fMan : REAL := 100;  (* PID varme rom. Manuelt kjoeling *)
    LH601_PID : fbSE_PID;  (* PID varme rom *)
    LH601_PID_Kp : REAL := 1;  (* PID varme rom. Forsterkning *)
    LH601_PID_Ti : REAL := 10;  (* PID varme rom. I-tid *)
    LH601_PID_Td : REAL;  (* PID varme rom. D-tid *)
    LH601_PID_fMan : REAL := 100;  (* PID varme rom. Manuelt paadrag *)
    LH601_T : fbSE_Hyst;  (* Termostat varme rom *)
    LH601_T_On : REAL := 0.5;
    LH601_T_Off : REAL := 0.1;
    LC601_PID : fbSE_PID;  (* PID kjoeling rom *)
    LC601_PID_Kp : REAL := 1;  (* PID kjoeling rom. Forsterkning *)
    LC601_PID_Ti : REAL := 10;  (* PID kjoeling rom. I-tid *)
    LC601_PID_Td : REAL;  (* PID kjoeling rom. D-tid *)
    LC601_PID_fMan : REAL := 100;  (* PID varme rom. Manuelt kjoeling *)
    LC601_T : fbSE_Hyst;  (* Termostat kjoeling rom *)
    LC601_T_On : REAL := 0.5;
    LC601_T_Off : REAL := 0.1;
  END_VAR
  VAR_OUTPUT
    RB600_HVAC : BOOL;
    RY600_CV : REAL;
    RY600_OP : REAL;
    LH601_OP : REAL;
    LH602_OP : REAL;
    LH601_CMD : BOOL;
    LH602_CMD : BOOL;
    LC601_OP : REAL;
    LC602_OP : REAL;
    LC601_CMD : BOOL;
    LC602_CMD : BOOL;
  END_VAR
  VAR  (* added by the conversion: wires and edge detectors of the diagram *)
    _ADD13_OUT : REAL;
    _DIV22_ENO : BOOL;
    _DIV22_OUT : REAL;
  END_VAR

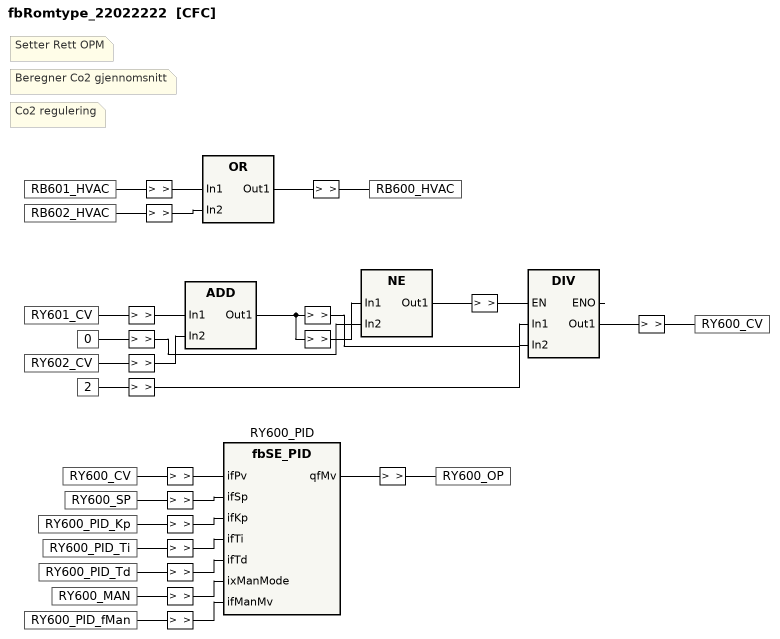
(* CFC diagram, written out as Structured Text *)
(* Setter Rett OPM *)
RB600_HVAC := RB601_HVAC OR RB602_HVAC;
(* Beregner Co2 gjennomsnitt *)
_ADD13_OUT := RY601_CV + RY602_CV;
_DIV22_OUT := DIV(EN := _ADD13_OUT <> 0, IN1 := _ADD13_OUT, IN2 := 2, ENO => _DIV22_ENO);
IF _DIV22_ENO THEN RY600_CV := _DIV22_OUT; END_IF;
(* Co2 regulering *)
RY600_PID(ifPv := RY600_CV, ifSp := RY600_SP, ifKp := RY600_PID_Kp, ifTi := RY600_PID_Ti, ifTd := RY600_PID_Td, ixManMode := RY600_MAN, ifManMv := RY600_PID_fMan);
RY600_OP := RY600_PID.qfMv;
END_FUNCTION_BLOCK

FUNCTION_BLOCK fbSE_Hyst
  VAR_INPUT
    rIn : REAL;
    rOn : REAL;
    rOff : REAL;
  END_VAR
  VAR_OUTPUT
    xOut : BOOL;
  END_VAR

					xOut:= ((rOn > rOff AND (rIn >= rOn OR (xOut AND rIn > rOff)))	OR		(rOn <rOff AND (rIn <= rOn OR (xOut AND rIn <rOff))));
				
END_FUNCTION_BLOCK

FUNCTION_BLOCK fbSE_PID
  VAR_INPUT
    ifPv : REAL;  (* Prosessvariabel (actual) *)
    ifSp : REAL;  (* Settpunkt *)
    ifKp : REAL := 1;  (* Forsterkning *)
    ifTi : REAL := 10;  (* I-tid *)
    ifTd : REAL;  (* D-tid *)
    ifBias : REAL;  (* Bias (Statisk paadrag som alltid er der) 0-100% *)
    ifInZero : REAL;  (* Nullpunkt for inn-verdi (PV og SP) *)
    ifInMax : REAL := 100;  (* Toppunkt for inn-verdi (PV og SP) *)
    ifOutZero : REAL;  (* Nullpunkt for ut-verdi (MV) *)
    ifOutMax : REAL := 100;  (* Toppunkt for ut-verdi (MV) *)
    ixManMode : BOOL;  (* Sender ManMv som MV, og resetter I-ledd *)
    ifManMv : REAL;  (* Manuelt paadrag som brukes i Man mode *)
  END_VAR
  VAR
    fPv : REAL;  (* Skalert PV (0-100) *)
    fSp : REAL;  (* Skalert SP (0-100) *)
    eRun : R_TRIG;  (* Resetter I-ledd ved endring rising edge i start betingelser *)
    fAvvik : REAL;  (* Avvik (Error) *)
    tCycleTimer : TON := (PT := TIME#1s0ms);  (* Teller syklus tiden *)
    fCycleTime : REAL;  (* Syklus tid i real *)
    fPID : REAL;  (* PID resultat (0-100%) *)
    fLastKp : REAL;  (* Forsterkning sist syklus (brukes til skalering ved endring) *)
    fLastTi : REAL;  (* Ti sist syklus (brukes til skalering ved endring) *)
    fLastIntegMax : REAL;  (* Max integral verdi sist syklus *)
    fIntegMax : REAL;  (* Max integral verdi (beregnet med Ti) *)
    fIntegral : REAL;  (* Integral verdi *)
    fI : REAL;  (* Integralt avvik *)
    fLastAvvik : REAL;  (* Avvik sist syklus *)
    fDerivat : REAL;  (* Derivat verdi *)
    fD : REAL;  (* Derivert avvik *)
  END_VAR
  VAR_OUTPUT
    qfMv : REAL;  (* Manipulert verdi (Resultat av PID) *)
    qxError : BOOL;  (* Feil alarm *)
  END_VAR

					eRun(CLK:= (ifKp > 0 AND NOT ixManMode));

IF ixManMode THEN																//Skriver manuelt SP til utgang
	qfMv := ifManMv;
ELSIF eRun.Q THEN																//Hvis det er rising edge paastart betingelser vil diverse variabler resettes/initializes
	fIntegral := 0;
	fIntegMax:= fLastIntegMax := 1 / ifKp * (100 / (1 / ifTi));
	fLastTi:= ifTi;
	fLastKp:= ifKp;
	fLastAvvik:= fAvvik;
	tCycleTimer(IN:= FALSE);
	tCycleTimer(IN:= TRUE);
ELSIF ifKp > 0 THEN												//Hvis Kp er satt, kjoeres PID funksjon

	//Felles
		IF(ifInMax - ifInZero) = 0 THEN											//Sjekker om vi deler paa 0, og gir ut evt. feil
		qxError := TRUE;
		RETURN;
	ELSE																		//	Ellers omskaleres Inn-verdier fra valgt til 0-100, og feil resettes
		qxError := FALSE;
		fPv:= (100 / (ifInMax - ifInZero)) * (ifPv - ifInZero);
		fSp:= (100 / (ifInMax - ifInZero)) * (ifSP - ifInZero);
	END_IF

	//Teller syklys tid
	tCycleTimer();																//Kjoerer TON for aa sjekke hvor lang tid som har gaatt siden forgje utregning
	fCycleTime:= 0.001 * TIME_TO_REAL(tCycleTimer.ET);							//Omskalerer syklus tid fra TIME til REAL
	tCycleTimer(IN:= FALSE);													//Resetter TON
	tCycleTimer(IN:= TRUE);


	//Proporsjonalt avvik
	fAvvik:= fSp - fPv;															//Beregner avvik som brukes i P-leddet


	//Integralt avvik
	IF ifTi > 0 THEN															//Hvis I er mer en 0, kjoerer vi I-ledd beregning
		IF ifTi <> fLastTi OR ifKp <> fLastKp THEN								//Hvis Ti eller Kp endrer seg, omskaleres max verdi for integral og den eksisterende integral verdien. Lagrer div variabler til neste sjekk/skalering
			fIntegMax := 1 / ifKp * (100 / (1 / ifTi));
			fIntegral:= (fIntegMax / fLastIntegMax) * fIntegral;
			fLastIntegMax:= fIntegMax;
			fLastTi:= ifTi;
			fLastKp:= ifKp;
		END_IF

		fIntegral := LIMIT(0, (fIntegral + fAvvik * fCycleTime), fIntegMax);		//Beregner integral

		fI:= (1 / ifTi) * fIntegral;												//Beregner I-verdien

	ELSE
		fI := 0;																	//Skriver i til 0 hvis Ti er 0
	END_IF

	//Derivert avvik
	IF(fAvvik - fLastAvvik)<> 0  AND ifTd > 0 THEN							//Sjekker om D-ledd er i bruk, og hindrer at vi deler paa 0 ved feil
		fDerivat := (fAvvik - fLastAvvik) / fCycleTime;							//Deriverer avviket
		fD:= LIMIT(-100, (ifTd * fDerivat), 100);								//Beregner D-verdien
	ELSE
		fD := 0;
	END_IF


	//PID utregnign
	fPID:= LIMIT(0, (ifKp * (fAvvik + fI + fD) + ifBias), 100);				//Beregner PID utverdi i 0-100

	IF(ifOutMax - ifOutZero) = 0 THEN											//Sjekker om vi deler paa 0
		qxError := TRUE;
	ELSE																		//	Hvis ikke, omskaleres ut signal til valgt span og feil resettes
		qxError := FALSE;
		qfMv:= ((ifOutMax - ifOutZero) / 100) * fPID + ifOutZero;
	END_IF

ELSE																			//Skriver utgang til 0, hvis PID ikke er paa
	qfMv := 0;
END_IF
				
END_FUNCTION_BLOCK

PROGRAM PRG_KNX_563_1
  VAR
    i : INT := 0;  (* Felles *)
    Interval : TON := (PT := TIME#2m0s0ms);
    typDPT : typDPT;
    KNX_master_1 : WagoAppKNX.FbKNX_Master;  (* Master *)
    M1_001_001_RB601_V : fbDPT_Switch_pro;  (* 001 *)
    M1_002_001_RB601_HVAC : fbDPT_Switch_pro;
    M1_003_001_RT601_CT : fbDPT_Value_Temp_pro;
    M1_004_001_RY601_CV : fbDPT_Value_AirQuality_pro;
    M1_005_001_LH601_OP : fbDPT_Scaling_pro;
    M1_006_001_LH601_CMD : fbDPT_Switch_pro;
    M1_007_001_LC601_OP : fbDPT_Scaling_pro;
    M1_008_001_LC601_CMD : fbDPT_Switch_pro;
    M1_009_002_RB601_V : fbDPT_Switch_pro;  (* 002 *)
    M1_0010_002_RB602_V : fbDPT_Switch_pro;
    M1_011_002_RB601_HVAC : fbDPT_Switch_pro;
    M1_012_002_RB602_HVAC : fbDPT_Switch_pro;
    M1_013_002_RT601_CT : fbDPT_Value_Temp_pro;
    M1_014_002_RY601_CV : fbDPT_Value_AirQuality_pro;
    M1_015_002_LH601_OP : fbDPT_Scaling_pro;
    M1_016_002_LH601_CMD : fbDPT_Switch_pro;
    M1_017_002_LC601_OP : fbDPT_Scaling_pro;
    M1_018_002_LC601_CMD : fbDPT_Switch_pro;
    M1_019_003_RB601_V : fbDPT_Switch_pro;  (* 003 *)
    M1_020_003_RB601_HVAC : fbDPT_Switch_pro;
    M1_021_003_RT601_CT : fbDPT_Value_Temp_pro;
    M1_022_003_RT602_CT : fbDPT_Value_Temp_pro;
    M1_023_003_RY601_CV : fbDPT_Value_AirQuality_pro;
    M1_024_003_LH601_OP : fbDPT_Scaling_pro;
    M1_025_003_LH601_CMD : fbDPT_Switch_pro;
    M1_026_003_LC601_OP : fbDPT_Scaling_pro;
    M1_027_003_LC601_CMD : fbDPT_Switch_pro;
    M1_028_004_RB601_V : fbDPT_Switch_pro;  (* 004 *)
    M1_029_004_RB601_HVAC : fbDPT_Switch_pro;
    M1_030_004_RT601_CT : fbDPT_Value_Temp_pro;
    M1_031_004_RY601_CV : fbDPT_Value_AirQuality_pro;
    M1_032_004_RY602_CV : fbDPT_Value_AirQuality_pro;
    M1_033_004_LH601_OP : fbDPT_Scaling_pro;
    M1_034_004_LH601_CMD : fbDPT_Switch_pro;
    M1_035_004_LC601_OP : fbDPT_Scaling_pro;
    M1_036_004_LC601_CMD : fbDPT_Switch_pro;
    M1_037_005_RB601_V : fbDPT_Switch_pro;  (* 005 *)
    M1_038_005_RB601_HVAC : fbDPT_Switch_pro;
    M1_039_005_RT601_CT : fbDPT_Value_Temp_pro;
    M1_040_005_RY601_CV : fbDPT_Value_AirQuality_pro;
    M1_041_005_LH601_OP : fbDPT_Scaling_pro;
    M1_042_005_LH602_OP : fbDPT_Scaling_pro;
    M1_043_005_LH601_CMD : fbDPT_Switch_pro;
    M1_044_005_LC601_OP : fbDPT_Scaling_pro;
    M1_045_005_LC601_CMD : fbDPT_Switch_pro;
    M1_046_006_RB601_V : fbDPT_Switch_pro;  (* 006 *)
    M1_047_006_RB601_HVAC : fbDPT_Switch_pro;
    M1_048_006_RT601_CT : fbDPT_Value_Temp_pro;
    M1_049_006_RY601_CV : fbDPT_Value_AirQuality_pro;
    M1_050_006_LH601_OP : fbDPT_Scaling_pro;
    M1_051_006_LH601_CMD : fbDPT_Switch_pro;
    M1_052_006_LH602_CMD : fbDPT_Switch_pro;
    M1_053_006_LC601_OP : fbDPT_Scaling_pro;
    M1_054_006_LC601_CMD : fbDPT_Switch_pro;
    M1_055_007_RB601_V : fbDPT_Switch_pro;  (* 007 *)
    M1_056_007_RB601_HVAC : fbDPT_Switch_pro;
    M1_057_007_RT601_CT : fbDPT_Value_Temp_pro;
    M1_058_007_RY601_CV : fbDPT_Value_AirQuality_pro;
    M1_059_007_LH601_OP : fbDPT_Scaling_pro;
    M1_060_007_LH601_CMD : fbDPT_Switch_pro;
    M1_061_007_LC601_OP : fbDPT_Scaling_pro;
    M1_062_007_LC602_OP : fbDPT_Scaling_pro;
    M1_063_007_LC601_CMD : fbDPT_Switch_pro;
    M1_064_008_RB601_V : fbDPT_Switch_pro;  (* 008 *)
    M1_065_008_RB601_HVAC : fbDPT_Switch_pro;
    M1_066_008_RT601_CT : fbDPT_Value_Temp_pro;
    M1_067_008_RY601_CV : fbDPT_Value_AirQuality_pro;
    M1_068_008_LH601_OP : fbDPT_Scaling_pro;
    M1_069_008_LH601_CMD : fbDPT_Switch_pro;
    M1_070_008_LC601_OP : fbDPT_Scaling_pro;
    M1_071_008_LC601_CMD : fbDPT_Switch_pro;
    M1_072_008_LC602_CMD : fbDPT_Switch_pro;
    M1_073_009_RB601_V : fbDPT_Switch_pro;  (* 009 *)
    M1_074_009_RB601_HVAC : fbDPT_Switch_pro;
    M1_075_009_RT601_CT : fbDPT_Value_Temp_pro;
    M1_076_009_RT602_CT : fbDPT_Value_Temp_pro;
    M1_077_009_RY601_CV : fbDPT_Value_AirQuality_pro;
    M1_078_009_LH601_OP : fbDPT_Scaling_pro;
    M1_079_009_LH602_OP : fbDPT_Scaling_pro;
    M1_080_009_LH601_CMD : fbDPT_Switch_pro;
    M1_081_009_LC601_OP : fbDPT_Scaling_pro;
    M1_082_009_LC601_CMD : fbDPT_Switch_pro;
    M1_083_010_RB601_V : fbDPT_Switch_pro;  (* 010 *)
    M1_084_010_RB601_HVAC : fbDPT_Switch_pro;
    M1_085_010_RT601_CT : fbDPT_Value_Temp_pro;
    M1_086_010_RT602_CT : fbDPT_Value_Temp_pro;
    M1_087_010_RY601_CV : fbDPT_Value_AirQuality_pro;
    M1_088_010_LH601_OP : fbDPT_Scaling_pro;
    M1_089_010_LH601_CMD : fbDPT_Switch_pro;
    M1_090_010_LH602_CMD : fbDPT_Switch_pro;
    M1_091_010_LC601_OP : fbDPT_Scaling_pro;
    M1_092_010_LC601_CMD : fbDPT_Switch_pro;
    M1_093_011_RB601_V : fbDPT_Switch_pro;  (* 011 *)
    M1_094_011_RB601_HVAC : fbDPT_Switch_pro;
    M1_095_011_RT601_CT : fbDPT_Value_Temp_pro;
    M1_096_011_RT602_CT : fbDPT_Value_Temp_pro;
    M1_097_011_RY601_CV : fbDPT_Value_AirQuality_pro;
    M1_098_011_LH601_OP : fbDPT_Scaling_pro;
    M1_099_011_LH601_CMD : fbDPT_Switch_pro;
    M1_100_011_LC601_OP : fbDPT_Scaling_pro;
    M1_101_011_LC602_OP : fbDPT_Scaling_pro;
    M1_102_011_LC601_CMD : fbDPT_Switch_pro;
    M1_103_012_RB601_V : fbDPT_Switch_pro;  (* 012 *)
    M1_104_012_RB601_HVAC : fbDPT_Switch_pro;
    M1_105_012_RT601_CT : fbDPT_Value_Temp_pro;
    M1_106_012_RT602_CT : fbDPT_Value_Temp_pro;
    M1_107_012_RY601_CV : fbDPT_Value_AirQuality_pro;
    M1_108_012_LH601_OP : fbDPT_Scaling_pro;
    M1_109_012_LH601_CMD : fbDPT_Switch_pro;
    M1_110_012_LC601_OP : fbDPT_Scaling_pro;
    M1_111_012_LC601_CMD : fbDPT_Switch_pro;
    M1_112_012_LC602_CMD : fbDPT_Switch_pro;
    M1_113_013_RB601_V : fbDPT_Switch_pro;  (* 013 *)
    M1_114_013_RB601_HVAC : fbDPT_Switch_pro;
    M1_115_013_RT601_CT : fbDPT_Value_Temp_pro;
    M1_116_013_RT602_CT : fbDPT_Value_Temp_pro;
    M1_117_013_RY601_CV : fbDPT_Value_AirQuality_pro;
    M1_118_013_RY602_CV : fbDPT_Value_AirQuality_pro;
    M1_119_013_LH601_OP : fbDPT_Scaling_pro;
    M1_120_013_LH601_CMD : fbDPT_Switch_pro;
    M1_121_013_LC601_OP : fbDPT_Scaling_pro;
    M1_122_013_LC601_CMD : fbDPT_Switch_pro;
    M1_123_014_RB601_V : fbDPT_Switch_pro;  (* 014 *)
    M1_124_014_RB601_HVAC : fbDPT_Switch_pro;
    M1_125_014_RT601_CT : fbDPT_Value_Temp_pro;
    M1_126_014_RT602_CT : fbDPT_Value_Temp_pro;
    M1_127_014_RY601_CV : fbDPT_Value_AirQuality_pro;
    M1_128_014_RY602_CV : fbDPT_Value_AirQuality_pro;
    M1_129_014_LH601_OP : fbDPT_Scaling_pro;
    M1_130_014_LH602_OP : fbDPT_Scaling_pro;
    M1_131_014_LH601_CMD : fbDPT_Switch_pro;
    M1_132_014_LH602_CMD : fbDPT_Switch_pro;
    M1_133_014_LC601_OP : fbDPT_Scaling_pro;
    M1_134_014_LC602_OP : fbDPT_Scaling_pro;
    M1_135_014_LC601_CMD : fbDPT_Switch_pro;
    M1_136_014_LC602_CMD : fbDPT_Switch_pro;
    M1_137_015_RB601_V : fbDPT_Switch_pro;  (* 015 *)
    M1_138_015_RB602_V : fbDPT_Switch_pro;
    M1_139_015_RB601_HVAC : fbDPT_Switch_pro;
    M1_140_015_RB602_HVAC : fbDPT_Switch_pro;
    M1_141_015_RT601_CT : fbDPT_Value_Temp_pro;
    M1_142_015_RT602_CT : fbDPT_Value_Temp_pro;
    M1_143_015_RY601_CV : fbDPT_Value_AirQuality_pro;
    M1_144_015_RY602_CV : fbDPT_Value_AirQuality_pro;
    M1_145_015_LH601_OP : fbDPT_Scaling_pro;
    M1_146_015_LH602_OP : fbDPT_Scaling_pro;
    M1_147_015_LH601_CMD : fbDPT_Switch_pro;
    M1_148_015_LH602_CMD : fbDPT_Switch_pro;
    M1_149_015_LC601_OP : fbDPT_Scaling_pro;
    M1_150_015_LC602_OP : fbDPT_Scaling_pro;
    M1_151_015_LC601_CMD : fbDPT_Switch_pro;
    M1_152_015_LC602_CMD : fbDPT_Switch_pro;
    M1_153_016_RB601_V : fbDPT_Switch_pro;  (* 016 *)
    M1_154_016_RB602_V : fbDPT_Switch_pro;
    M1_155_016_RB601_HVAC : fbDPT_Switch_pro;
    M1_156_016_RB602_HVAC : fbDPT_Switch_pro;
    M1_157_016_RY601_CV : fbDPT_Value_AirQuality_pro;
    M1_158_016_RY602_CV : fbDPT_Value_AirQuality_pro;
    M1_159_016_LH601_OP : fbDPT_Scaling_pro;
    M1_160_016_LH602_OP : fbDPT_Scaling_pro;
    M1_161_016_LH601_CMD : fbDPT_Switch_pro;
    M1_162_016_LH602_CMD : fbDPT_Switch_pro;
    M1_163_016_LC601_OP : fbDPT_Scaling_pro;
    M1_164_016_LC602_OP : fbDPT_Scaling_pro;
    M1_165_016_LC601_CMD : fbDPT_Switch_pro;
    M1_166_016_LC602_CMD : fbDPT_Switch_pro;
  END_VAR
  VAR  (* added by the conversion: wires and edge detectors of the diagram *)
    _ADD9_OUT : INT;
    _GT15_OUT : BOOL;
    _MOVE19_ENO : BOOL;
    _MOVE19_OUT : INT;
    _MOVE46_ENO : BOOL;
    _MOVE46_OUT : ANY;
    _MOVE59_ENO : BOOL;
    _MOVE59_OUT : ANY;
    _MOVE72_ENO : BOOL;
    _MOVE72_OUT : ANY;
    _MOVE85_ENO : BOOL;
    _MOVE85_OUT : ANY;
    _MOVE163_ENO : BOOL;
    _MOVE163_OUT : ANY;
    _MOVE176_ENO : BOOL;
    _MOVE176_OUT : ANY;
    _MOVE189_ENO : BOOL;
    _MOVE189_OUT : ANY;
    _MOVE202_ENO : BOOL;
    _MOVE202_OUT : ANY;
    _MOVE215_ENO : BOOL;
    _MOVE215_OUT : ANY;
    _MOVE228_ENO : BOOL;
    _MOVE228_OUT : ANY;
    _MOVE306_ENO : BOOL;
    _MOVE306_OUT : ANY;
    _MOVE319_ENO : BOOL;
    _MOVE319_OUT : ANY;
    _MOVE332_ENO : BOOL;
    _MOVE332_OUT : ANY;
    _MOVE345_ENO : BOOL;
    _MOVE345_OUT : ANY;
    _MOVE358_ENO : BOOL;
    _MOVE358_OUT : ANY;
    _MOVE436_ENO : BOOL;
    _MOVE436_OUT : ANY;
    _MOVE449_ENO : BOOL;
    _MOVE449_OUT : ANY;
    _MOVE462_ENO : BOOL;
    _MOVE462_OUT : ANY;
    _MOVE475_ENO : BOOL;
    _MOVE475_OUT : ANY;
    _MOVE488_ENO : BOOL;
    _MOVE488_OUT : ANY;
    _MOVE566_ENO : BOOL;
    _MOVE566_OUT : ANY;
    _MOVE579_ENO : BOOL;
    _MOVE579_OUT : ANY;
    _MOVE592_ENO : BOOL;
    _MOVE592_OUT : ANY;
    _MOVE605_ENO : BOOL;
    _MOVE605_OUT : ANY;
    _MOVE699_ENO : BOOL;
    _MOVE699_OUT : ANY;
    _MOVE712_ENO : BOOL;
    _MOVE712_OUT : ANY;
    _MOVE725_ENO : BOOL;
    _MOVE725_OUT : ANY;
    _MOVE738_ENO : BOOL;
    _MOVE738_OUT : ANY;
    _MOVE832_ENO : BOOL;
    _MOVE832_OUT : ANY;
    _MOVE845_ENO : BOOL;
    _MOVE845_OUT : ANY;
    _MOVE858_ENO : BOOL;
    _MOVE858_OUT : ANY;
    _MOVE871_ENO : BOOL;
    _MOVE871_OUT : ANY;
    _MOVE965_ENO : BOOL;
    _MOVE965_OUT : ANY;
    _MOVE978_ENO : BOOL;
    _MOVE978_OUT : ANY;
    _MOVE991_ENO : BOOL;
    _MOVE991_OUT : ANY;
    _MOVE1004_ENO : BOOL;
    _MOVE1004_OUT : ANY;
    _MOVE1098_ENO : BOOL;
    _MOVE1098_OUT : ANY;
    _MOVE1111_ENO : BOOL;
    _MOVE1111_OUT : ANY;
    _MOVE1124_ENO : BOOL;
    _MOVE1124_OUT : ANY;
    _MOVE1137_ENO : BOOL;
    _MOVE1137_OUT : ANY;
    _MOVE1150_ENO : BOOL;
    _MOVE1150_OUT : ANY;
    _MOVE1244_ENO : BOOL;
    _MOVE1244_OUT : ANY;
    _MOVE1257_ENO : BOOL;
    _MOVE1257_OUT : ANY;
    _MOVE1270_ENO : BOOL;
    _MOVE1270_OUT : ANY;
    _MOVE1283_ENO : BOOL;
    _MOVE1283_OUT : ANY;
    _MOVE1296_ENO : BOOL;
    _MOVE1296_OUT : ANY;
    _MOVE1390_ENO : BOOL;
    _MOVE1390_OUT : ANY;
    _MOVE1403_ENO : BOOL;
    _MOVE1403_OUT : ANY;
    _MOVE1416_ENO : BOOL;
    _MOVE1416_OUT : ANY;
    _MOVE1429_ENO : BOOL;
    _MOVE1429_OUT : ANY;
    _MOVE1442_ENO : BOOL;
    _MOVE1442_OUT : ANY;
    _MOVE1536_ENO : BOOL;
    _MOVE1536_OUT : ANY;
    _MOVE1549_ENO : BOOL;
    _MOVE1549_OUT : ANY;
    _MOVE1562_ENO : BOOL;
    _MOVE1562_OUT : ANY;
    _MOVE1575_ENO : BOOL;
    _MOVE1575_OUT : ANY;
    _MOVE1588_ENO : BOOL;
    _MOVE1588_OUT : ANY;
    _MOVE1682_ENO : BOOL;
    _MOVE1682_OUT : ANY;
    _MOVE1695_ENO : BOOL;
    _MOVE1695_OUT : ANY;
    _MOVE1708_ENO : BOOL;
    _MOVE1708_OUT : ANY;
    _MOVE1721_ENO : BOOL;
    _MOVE1721_OUT : ANY;
    _MOVE1734_ENO : BOOL;
    _MOVE1734_OUT : ANY;
    _MOVE1747_ENO : BOOL;
    _MOVE1747_OUT : ANY;
    _MOVE1825_ENO : BOOL;
    _MOVE1825_OUT : ANY;
    _MOVE1838_ENO : BOOL;
    _MOVE1838_OUT : ANY;
    _MOVE1851_ENO : BOOL;
    _MOVE1851_OUT : ANY;
    _MOVE1864_ENO : BOOL;
    _MOVE1864_OUT : ANY;
    _MOVE1877_ENO : BOOL;
    _MOVE1877_OUT : ANY;
    _MOVE1890_ENO : BOOL;
    _MOVE1890_OUT : ANY;
    _MOVE2032_ENO : BOOL;
    _MOVE2032_OUT : ANY;
    _MOVE2045_ENO : BOOL;
    _MOVE2045_OUT : ANY;
    _MOVE2058_ENO : BOOL;
    _MOVE2058_OUT : ANY;
    _MOVE2071_ENO : BOOL;
    _MOVE2071_OUT : ANY;
    _MOVE2084_ENO : BOOL;
    _MOVE2084_OUT : ANY;
    _MOVE2097_ENO : BOOL;
    _MOVE2097_OUT : ANY;
    _MOVE2110_ENO : BOOL;
    _MOVE2110_OUT : ANY;
    _MOVE2123_ENO : BOOL;
    _MOVE2123_OUT : ANY;
    _MOVE2265_ENO : BOOL;
    _MOVE2265_OUT : ANY;
    _MOVE2278_ENO : BOOL;
    _MOVE2278_OUT : ANY;
    _MOVE2291_ENO : BOOL;
    _MOVE2291_OUT : ANY;
    _MOVE2304_ENO : BOOL;
    _MOVE2304_OUT : ANY;
    _MOVE2317_ENO : BOOL;
    _MOVE2317_OUT : ANY;
    _MOVE2330_ENO : BOOL;
    _MOVE2330_OUT : ANY;
  END_VAR

